//link encoder calibartion data
m_linkEncoderDir :=GVL_CartJointEncoderCaliData.g_asbEncoderDir[i_jntIdx];
m_minLinkEncoder :=GVL_CartJointEncoderCaliData.g_minLinkEncoder[ i_jntIdx] - m_linkEncoderDir*GVL_SetupJointEncoderCaliData.g_linkEncLimitBuffer; // expand limit
m_maxLinkEncoder :=GVL_CartJointEncoderCaliData.g_maxLinkEncoder[ i_jntIdx] + m_linkEncoderDir*GVL_SetupJointEncoderCaliData.g_linkEncLimitBuffer; // expand limit
m_caliLinkEncoder :=GVL_CartJointEncoderCaliData.g_caliLinkEncoder[ i_jntIdx];
m_linkEncCaliJntPos :=GVL_CartJointEncoderCaliData.g_linkEncCaliJntPos[i_jntIdx];
m_linkEncZeroCross :=GVL_CartJointEncoderCaliData.g_linkEncZeroCross[ i_jntIdx];
m_multiCycles :=GVL_CartJointEncoderCaliData.g_multipleCyclesJoint[i_jntIdx];

// convert cali link encoder if joint cross zero
IF 1=m_linkEncZeroCross THEN
	IF 1=m_linkEncoderDir AND m_caliLinkEncoder < m_minLinkEncoder THEN
		m_caliLinkEncoder := GVL_CartJointEncoderCaliData.g_caliLinkEncoder[ i_jntIdx] + m_linkEncoderRes;
	ELSIF -1=m_linkEncoderDir AND m_caliLinkEncoder < m_maxLinkEncoder THEN
		m_caliLinkEncoder := GVL_CartJointEncoderCaliData.g_caliLinkEncoder[ i_jntIdx] + m_linkEncoderRes;
	END_IF
END_IF

// macro data
m_trq2CurrentRatio:=m_motorDir * 1000.0/(m_trqConst*m_motorReduction);
m_current2TrqRatio:=m_motorDir * (m_trqConst*m_motorReduction)/1000.0;
m_linkEnc2PosRatio := 2*PI*m_linkEncoderDir/(m_linkEncoderReduction*m_linkEncoderRes);
m_motorEnc2PosRatio := 2*PI * m_motorDir/(m_motorReduction * m_motorEncoderRes);


// motor data init
m_rawJntVel :=0;
m_curJntVel:=0;
m_curJntTrq :=0;
m_rawCurrent :=0;
m_filtCurrent :=0;
m_cmdJntVel :=0.0;
m_cmdJntTrq :=0.0;
m_cmdCurrent := 0.0;

// filter init
m_jntVelLpf.init(1, GVL_CartControlParameters.g_curJntVelLpfCutoffFreq, g_cartCtrlFreq);
m_cmdTrqLpf.init(1, GVL_CartControlParameters.g_cmdJntTrqLpfCutoffFreq, g_cartCtrlFreq);
m_curTrqLpf.init(1, GVL_CartControlParameters.g_curJntTrqLpfCutoffFreq, g_cartCtrlFreq);

// driver init value
m_motorOutputs.m_controlWord:=DriverCtrlWord_INIT;
m_motorOutputs.m_opMode:=INT_TO_SINT(DriverOPMode_Pos);
m_motorOutputs.m_cmdCurrent:=0;
m_motorOutputs.m_cmdMotorEncoder:=m_motorInputs.m_motorEncoder;
END_METHOD

METHOD PUBLIC updateCmd : BOOL
VAR_INPUT
	i_opMode : E_DriverOPMode;
	i_cmdPos :LREAL;
	i_cmdTrq :LREAL;
	i_cmdVel :LREAL;
END_VAR
VAR
	i:INT;
END_VAR
m_motorOutputs.m_opMode:=INT_TO_SINT( i_opMode);

// pos mode
IF i_opMode = DriverOPMode_Pos OR i_opMode = DriverOPMode_cspMZ  THEN
	m_motorOutputs.m_cmdCurrent:=0;
	m_cmdJntPos :=i_cmdPos;
	m_motorOutputs.m_cmdMotorEncoder :=motorPos2Enc(m_cmdJntPos);
ELSIF i_opMode = DriverOPMode_Vel THEN
	m_cmdJntVel := i_cmdVel;
	m_cartMotorOutput.m_cmdVelMzVelMode := cmd2motorMZ(m_cmdJntVel, g_cartCtrlCycleTime);
ELSIF i_opMode = DriverOPMode_Trq THEN   //Here the torque mode is equal to the contour position mode of the MingZhi driver
	m_cmdJntVel := i_cmdVel;
	m_cmdAcc:=i_cmdVel*2;
	m_cmdJntPos:=i_cmdPos;
	m_cartMotorOutput.m_cmdAccMz :=cmd2motorMZ(m_cmdAcc, g_cartCtrlCycleTime);
	m_cartMotorOutput.m_cmdVelMz := cmd2motorMZ(m_cmdJntVel, g_cartCtrlCycleTime);
	m_motorOutputs.m_cmdMotorEncoder := motorPos2Enc(m_cmdJntVel);
ELSIF i_opMode = DriverOPMode_csvMZ THEN
	m_cmdJntVel := i_cmdVel;
	m_cartMotorOutput.m_cmdVelMzVelMode := cmd2motorMZ(m_cmdJntVel, g_cartCtrlCycleTime);
END_IF
END_METHOD

METHOD PUBLIC updateStatus : BOOL
VAR_INPUT
END_VAR
// compute joint position
m_curLinkPos:= linkEnc2Pos();
m_curMotorPos:=motorEnc2Pos();
m_curLinkSingle := m_curLinkPos - 2*PI* m_linkEncCycles;

// Cart joint1-4 have no link enconder, use motor position
IF m_jntIdx <= 4 THEN
	m_curJntPos := m_curMotorPos;
ELSE
	m_curJntPos := m_curLinkPos;
END_IF

// compute joint velocity
m_curVelCalCycles := m_curVelCalCycles+1;
IF m_curVelCalCycles > m_velCalcCycles THEN
	m_rawJntVel:= (m_curJntPos-m_lastJntPos)/(m_cycleTime*m_velCalcCycles);
	m_curJntVel := m_jntVelLpf.run(m_rawJntVel);
	m_lastJntPos :=m_curJntPos;	
	m_curVelCalCycles:=1;
END_IF


// current and torque
m_rawCurrent := m_motorInputs.m_current;
m_filtCurrent := m_curTrqLpf.run(m_rawCurrent);
m_curJntTrq := m_filtCurrent * m_current2TrqRatio;
END_METHOD

END_FUNCTION_BLOCK

// ---- FBs_Robots/FB_JointBase.TcPOU
FUNCTION_BLOCK FB_JointBase
VAR_INPUT
END_VAR
VAR_OUTPUT
END_VAR
VAR
	// arm and joint index
	m_armIdx :INT;
	m_jntIdx :INT;
	
	// motor IO
	m_motorInputs AT%I*	:ST_MotorInputs;
	m_motorOutputs AT%Q* :ST_MotorOutputs;
	
	// cycle time
	m_cycleTime :LREAL;
	
	// calibrated link encoder data
	m_minLinkEncoder :DINT;
	m_maxLinkEncoder :DINT;
	m_caliLinkEncoder :DINT;
	m_linkEncCaliJntPos :LREAL;
	m_linkEncZeroCross :INT;
	m_initMotorEnc : DINT;
	m_multiCycles :INT;
	
	// joint position from link encoder after power on
	m_initLinkPos :LREAL;
	
	// data for link encoder multiple cycles
	m_lastLinkEncoder :DINT;
	m_linkEncCycles:INT;
	
	// device paramters
	m_motorEncoderRes :DINT;
	m_linkEncoderRes :DINT;
	m_motorReduction :LREAL;
	m_linkEncoderReduction :LREAL;
	m_trqConst :LREAL;
	m_maxCurrent :LREAL;
	m_motorDir :INT;								
	m_linkEncoderDir :INT;
	m_minJntPos: LREAL;
	m_maxJntPos: LREAL;
	
	// macro defined data for quick calculation
	m_trq2CurrentRatio:LREAL;
	m_current2TrqRatio:LREAL;
	m_linkEnc2PosRatio :LREAL;
	m_motorEnc2PosRatio :LREAL;
	
	// joint data
	m_curMotorPos :LREAL;
	m_curLinkPos :LREAL;
	m_curLinkSingle :LREAL;//[0-360]
	m_curJntPos	:LREAL;
	m_curJntVel :LREAL;
	m_rawJntVel :LREAL;
	m_curJntTrq :	LREAL;
	m_rawCurrent : LREAL;
	m_filtCurrent : LREAL;
	m_cmdJntPos :LREAL;
	m_cmdJntVel :LREAL;
	m_cmdJntTrq :LREAL;
	m_cmdCurrent : LREAL;
	m_lastJntPos :LREAL;
	
	// velocity filter
	m_jntVelLpf :FB_LowPassFilter;
	
	// command torque filter
	m_curTrqLpf : FB_LowPassFilter;
	m_cmdTrqLpf :FB_LowPassFilter;
	
	// velocity is calculated every (m_velCalcCycles) control cycles
	// TODO: insturment joint motor can not reach 4k now, so calculate their velocity with 1k frequency, need to remove later
	m_velCalcCycles :INT :=1;
	m_curVelCalCycles :INT :=1;
	
	// SDO writer
	m_opModeSDOWrite:FB_EcCoESdoWrite;
	m_MotorCurrentSDOWrite:FB_EcCoESdoWrite;
	
END_VAR

PROPERTY cmdCurrent : LREAL
GET
cmdCurrent:=m_cmdCurrent;
END_GET
END_PROPERTY

METHOD PUBLIC disable : BOOL
VAR_INPUT
END_VAR
m_motorOutputs.m_controlWord:=DriverCtrlWord_INIT;
disable:=true;
END_METHOD

METHOD PUBLIC enable : BOOL
VAR_INPUT
END_VAR
IF DriverStatusWord_INIT = m_motorInputs.m_statusWord THEN
	m_motorOutputs.m_controlWord:=DriverCtrlWord_PREOP;
	enable := FALSE;
ELSIF DriverStatusWord_PREOP = m_motorInputs.m_statusWord THEN
	m_motorOutputs.m_controlWord:=DriverCtrlWord_OP;
	enable :=  FALSE;
ELSIF DriverStatusWord_OP = m_motorInputs.m_statusWord THEN
	enable :=  TRUE;
//ELSE
//	m_motorOutputs.m_controlWord:=DriverCtrlWord_INIT;
//	enable :=  FALSE;
END_IF
END_METHOD

PROPERTY filtCurrent : LREAL
GET
filtCurrent:=m_filtCurrent;
END_GET
END_PROPERTY

METHOD PUBLIC initJntPos : BOOL
VAR_INPUT
END_VAR
m_lastLinkEncoder :=m_motorInputs.m_linkEncoder;
m_linkEncCycles:=0;
m_curLinkPos :=linkEnc2Pos();
m_initLinkPos:=m_curLinkPos;
m_initMotorEnc :=m_motorInputs.m_motorEncoder;
m_curMotorPos:=motorEnc2Pos();
m_curJntPos := m_curMotorPos;
m_cmdJntPos :=m_curJntPos;	
m_lastJntPos :=m_curJntPos;
END_METHOD

PROPERTY initLinkPos : lreal
GET
initLinkPos:=m_initLinkPos;
END_GET
SET
m_initLinkPos:=initLinkPos;
END_SET
END_PROPERTY

METHOD PUBLIC isEnabled : BOOL
VAR_INPUT
END_VAR
isEnabled :=(DriverStatusWord_OP = m_motorInputs.m_statusWord);
END_METHOD

PROPERTY jntPos : LREAL
GET
jntPos := m_curJntPos;
END_GET
END_PROPERTY

PROPERTY jntTrq : LREAL
GET
jntTrq:=m_curJntTrq;
END_GET
END_PROPERTY

PROPERTY jntVel : LREAL
GET
jntVel := m_curJntVel;
END_GET
END_PROPERTY

METHOD PROTECTED linkEnc2Pos : LREAL
VAR_INPUT
END_VAR
VAR
	incLinkPos :LREAL;
	newLinkEnc :DINT;
END_VAR
// cycle check
IF 1=m_multiCycles THEN
	IF (m_motorInputs.m_linkEncoder - m_lastLinkEncoder)*m_linkEncoderDir < -m_linkEncoderRes/2 THEN
		m_linkEncCycles :=m_linkEncCycles+1;
	ELSIF (m_motorInputs.m_linkEncoder - m_lastLinkEncoder)*m_linkEncoderDir > m_linkEncoderRes/2 THEN
		m_linkEncCycles :=m_linkEncCycles-1;
	END_IF
END_IF
m_lastLinkEncoder:=m_motorInputs.m_linkEncoder;

// convert link encoder if joint cross zero
newLinkEnc := m_motorInputs.m_linkEncoder;
IF 1=m_linkEncZeroCross AND 0 = m_multiCycles THEN
	IF 1=m_linkEncoderDir AND m_motorInputs.m_linkEncoder < m_minLinkEncoder THEN
		newLinkEnc := m_motorInputs.m_linkEncoder + m_linkEncoderRes;
	ELSIF -1=m_linkEncoderDir AND m_motorInputs.m_linkEncoder < m_maxLinkEncoder THEN
		newLinkEnc := m_motorInputs.m_linkEncoder + m_linkEncoderRes;
	END_IF
END_IF

// motion from calibrated points
incLinkPos := (newLinkEnc-m_caliLinkEncoder)*m_linkEnc2PosRatio;

// absolute joint position
linkEnc2Pos := incLinkPos + m_linkEncCaliJntPos + 2*PI* m_linkEncCycles;
END_METHOD

PROPERTY PUBLIC linkPos : LREAL
GET
linkPos:=m_curLinkPos;
END_GET
END_PROPERTY

PROPERTY linkSingle : LREAL
GET
linkSingle :=m_curLinkSingle;
END_GET
END_PROPERTY

METHOD PROTECTED motorEnc2Pos : LREAL
VAR_INPUT
END_VAR
motorEnc2Pos:= (m_motorInputs.m_motorEncoder-m_initMotorEnc)* m_motorEnc2PosRatio +m_initLinkPos;
END_METHOD

PROPERTY PUBLIC motorPos : LREAL
GET
motorPos := m_curMotorPos;
END_GET
END_PROPERTY

METHOD PROTECTED motorPos2Enc : DINT
VAR_INPUT
	i_jntPos :LREAL;
END_VAR

VAR
END_VAR
motorPos2Enc := LREAL_TO_DINT((i_jntPos-m_initLinkPos)/m_motorEnc2PosRatio + m_initMotorEnc);
END_METHOD

PROPERTY rawCurrent : LREAL
GET
rawCurrent := m_rawCurrent;
END_GET
END_PROPERTY

METHOD PROTECTED singleCyclePos : LREal
VAR_INPUT
END_VAR
VAR
	cycles :lreal;
END_VAR
cycles := ABS(FLOOR( m_curJntPos/g_2pi));
IF m_curJntPos<0 THEN
	singleCyclePos := m_curJntPos+cycles*g_2pi;
ELSE
	singleCyclePos := m_curJntPos-cycles*g_2pi;
END_IF
END_METHOD

METHOD PUBLIC updateCmds : BOOL
VAR_INPUT
	i_opMode : E_DriverOPMode;
	i_cmdPos :LREAL;
	i_cmdTrq :LREAL;
END_VAR
VAR
	filtCmdTrq :LREAL;
END_VAR
m_motorOutputs.m_opMode:=INT_TO_SINT( i_opMode);
// pos mode
IF i_opMode = DriverOPMode_Pos THEN
	m_motorOutputs.m_cmdCurrent:=0;
	m_cmdTrqLpf.reset();	
//	i_cmdPos:=LIMIT(m_minJntPos, i_cmdPos, m_maxJntPos); // May cause position jump, Do this in safety check. 
	m_cmdJntPos :=i_cmdPos;
	m_motorOutputs.m_cmdMotorEncoder :=motorPos2Enc(m_cmdJntPos);
ELSIF i_opMode = DriverOPMode_Trq THEN
	filtCmdTrq:=m_cmdTrqLpf.run(i_cmdTrq);
	m_motorOutputs.m_cmdCurrent:=LREAL_TO_DINT(LIMIT(-m_maxCurrent, filtCmdTrq*m_trq2CurrentRatio,m_maxCurrent));
	m_motorOutputs.m_cmdMotorEncoder :=m_motorInputs.m_motorEncoder; 
END_IF
m_cmdCurrent:=m_motorOutputs.m_cmdCurrent;
END_METHOD

METHOD PUBLIC updateStatus : BOOL
VAR_INPUT
END_VAR
// compute joint position
m_curLinkPos:= linkEnc2Pos();
m_curMotorPos:=motorEnc2Pos();
m_curJntPos := m_curMotorPos;
m_curLinkSingle := singleCyclePos();

// compute joint velocity
m_curVelCalCycles := m_curVelCalCycles+1;
IF m_curVelCalCycles > m_velCalcCycles THEN
	m_rawJntVel:= (m_curJntPos-m_lastJntPos)/(m_cycleTime*m_velCalcCycles);
	m_curJntVel := m_jntVelLpf.run(m_rawJntVel);
	m_lastJntPos :=m_curJntPos;	
	m_curVelCalCycles:=1;
END_IF


// current and torque
m_rawCurrent := m_motorInputs.m_current;
m_filtCurrent := m_curTrqLpf.run(m_rawCurrent);
m_curJntTrq := m_filtCurrent * m_current2TrqRatio;
END_METHOD

END_FUNCTION_BLOCK

// ---- FBs_CartControlles/FB_CartCtrlMotionCar.TcPOU
FUNCTION_BLOCK FB_CartCtrlMotionCar EXTENDS FB_CartCtrlBase
VAR_INPUT
END_VAR
VAR_OUTPUT
END_VAR
VAR
	m_driveForce: ARRAY [1..2] OF LREAL;
	
	// input drive force filter
	m_driveVelLpf : ARRAY [1..2] OF FB_LowPassFilter;
	m_driveForceFilter: Vec2i;
	
	//cart motion trajectory velocity
	m_trajVel : ARRAY [1..2] OF LREAL;
	m_motorDir :ARRAY [1..2] OF INT := [1,-1];
	
	m_tarJntPos : ARRAY [1..2] OF LREAL;
	m_incJntPos : ARRAY [1..2] OF LREAL;
	m_initJntPos : ARRAY [1..2] OF LREAL;
	// time threshold to drive wheel after it's enabled
	m_cartWheelDriveWaitTime :LREAL := 0.2;
	
	//wheel motion  time 
	m_wheelMotionTime:ARRAY [1..2] OF LREAL;
	
	// filter cut-off frequency for cart drive force 
	m_cmdJntVelLpfCutoffFreq : LREAL :=5;
END_VAR

VAR CONSTANT
	//Proportionality constant of force sensor
	m_driveForceProConstant : LREAL := 5/15000;
END_VAR

// override this function in each exact controller
METHOD PROTECTED calcCmdJntPos : BOOL
VAR_IN_OUT CONSTANT
	// slave cart joint data
	i_slaveCart :FB_SlaveCart;
END_VAR

VAR
	i:INT;
END_VAR

FOR i := 1 TO 2 BY 1 DO
	m_driveForce[i] :=LIMIT(-5, i_slaveCart.m_driveForce[i]/3000, 5);
	m_wheelMotionTime[i] := LIMIT(0, m_wheelMotionTime[i] + g_cartCtrlCycleTime, 1);
	
	IF m_wheelMotionTime[i] > m_cartWheelDriveWaitTime THEN
		m_trajVel[i] := m_driveVelLpf[i].run(i_rawData:=m_motorDir[i] * m_driveForce[i]/2);
		m_incJntPos[i] := m_incJntPos[i] + m_trajVel[i] * g_cartCtrlCycleTime;
		
		m_cmdJntPos[i+2] := m_initJntPos[i] + m_incJntPos[i];
	END_IF
END_FOR
END_METHOD

// override this function in each exact controller
// NOTICE: set joint control mode here, and do some initialization if needed
METHOD PUBLIC init : BOOL
VAR_IN_OUT CONSTANT
	i_slaveCart	:FB_SlaveCart;
END_VAR
VAR_IN_OUT 
	r_cartCtrlCmd :ST_SlaveArmCtrlCmds;
END_VAR
SUPER^.init(i_slaveCart,r_cartCtrlCmd);

m_jntEnableFlag[3] :=1;
m_jntEnableFlag[4] :=1;

m_jntOPMode[3]:= DriverOPMode_cspMZ;
m_jntOPMode[4]:= DriverOPMode_cspMZ;

m_tarJntPos[1] := 0;
m_tarJntPos[2] := 0;

m_incJntPos[1] := 0;
m_incJntPos[2] := 0;

m_initJntPos[1] := i_slaveCart.curJntPos[3];
m_initJntPos[2] := i_slaveCart.curJntPos[4];

m_driveVelLpf[1].init(i_filterOrd:= 1, i_cutoffFreq:= m_cmdJntVelLpfCutoffFreq, i_sampleFreq:= 8000);
m_driveVelLpf[2].init(i_filterOrd:= 1, i_cutoffFreq:= m_cmdJntVelLpfCutoffFreq, i_sampleFreq:= 8000);

m_driveVelLpf[1].run(i_rawData:=0);
m_driveVelLpf[2].run(i_rawData:=0);


m_wheelMotionTime[1]:=0;
m_wheelMotionTime[2]:=0;

// update commands to arm
copyCmds(r_cartCtrlCmd);
END_METHOD

END_FUNCTION_BLOCK

// ---- FBs_CartControlles/FB_CartCtrlAdjust.TcPOU
FUNCTION_BLOCK FB_CartCtrlAdjust EXTENDS FB_CartCtrlBase
VAR_INPUT
END_VAR
VAR_OUTPUT
END_VAR
VAR

	m_joystickSignal: Vec8d;	
	m_fiducialValue:INT:= 512;
	m_joystickRange:INT:=430;
	m_joystickDir: Vec8i:=[1,1,1,1,-1,-1,1,-1];
	m_joystickVelInc: Vec8d;
	m_actJntPos: Vec8d;
	m_tarPosInc: Vec8d;
	m_tarCartPos: Vec8d;
	m_trajJntPos : Vec8d;
	m_tarJntPos : Vec8d;
	m_initActJntPos: Vec8d;
	m_initActCartPos: Vec8d;
	m_veiwAngle : LREAL;

	m_carJntSoftwareLimit :ARRAY [5..8] OF LREAL := [0.005, 2*g_deg2Rad, 0.005, 2*g_deg2Rad];
	// input joystick signal filter
	m_joystickSignalLpf : ARRAY [1..4] OF FB_LowPassFilter;
	m_joystickSignalFilter: Vec8d;
	
	// time threshold to 5-8joint after it's enabled
	m_cartAdjustStartWaitTime :LREAL := 0.2;
	
	//adjust start  time 
	m_adjustStartTime :LREAL;
	
	// filter cut-off frequency for cart drive force 
	m_cmdJoystickLpfCutoffFreq : LREAL :=8;
	m_cartCtrlFreq :LREAL:=8000;
	
	m_jntOTG :ARRAY[1..8] OF FB_secOrdTrajFilter;
END_VAR

// override this function in each exact controller
METHOD PROTECTED calcCmdJntPos : BOOL
VAR_IN_OUT CONSTANT
	// slave cart joint data
	i_slaveCart :FB_SlaveCart;
END_VAR

VAR
	i:INT;
END_VAR
//In this method, 5 represents the pillar postion , 6 represents the beam rotation angle ,7 represents the beam stretch position ,8 represents the overhang angle
m_adjustStartTime :=LIMIT(0, m_adjustStartTime + g_cartCtrlCycleTime, 1);
m_actJntPos := i_slaveCart.curJntPos;
m_actJntPos[7] := i_slaveCart.curJntPos[7] + GVL_CartControlParameters.g_curBeamStretchJntInitPos;
m_veiwAngle := m_actJntPos[6] + m_actJntPos[8];

IF m_adjustStartTime > m_cartAdjustStartWaitTime THEN
	FOR i:= 1 TO 4 BY 1 DO
		m_joystickSignalFilter[i] := m_joystickSignalLpf[i].run(i_rawData:= m_joystickSignal[i]);
		m_joystickSignal[i] := i_slaveCart.m_joystickSignal[i] - m_fiducialValue;
		m_joystickVelInc[i+4] := m_joystickSignalFilter[i]/m_joystickRange*m_joystickDir[i+4]*GVL_CartControlParameters.g_maxCartVel[i];
		m_tarPosInc[i+4] := m_tarPosInc[i+4] + m_joystickVelInc[i+4] * g_cartCtrlCycleTime;
	END_FOR
	
	
	m_tarCartPos[5] := m_initActJntPos[5] + m_tarPosInc[5];
	IF i_slaveCart.m_ctrlEnable.camera_joysticks_enable THEN
		m_tarCartPos[6] := m_initActCartPos[6] + m_tarPosInc[6]*COS(m_veiwAngle)+m_tarPosInc[7]*SIN(m_veiwAngle);
		m_tarCartPos[7] := m_initActCartPos[7] - m_tarPosInc[6]*SIN(m_veiwAngle)+m_tarPosInc[7]*COS(m_veiwAngle);
	ELSE
		m_tarCartPos[6] := m_initActCartPos[6] + m_tarPosInc[6];
		m_tarCartPos[7] := m_initActCartPos[7] + m_tarPosInc[7];
	END_IF
	m_tarCartPos[8] := m_initActJntPos[8] + m_tarPosInc[8];
	
	IF i_slaveCart.m_ctrlEnable.limit_height_adjusting THEN
		m_trajJntPos[5] := m_tarCartPos[5];
	ELSE
		m_trajJntPos[5] := LIMIT(GVL_CartMotorParameters.g_minJntPos[5], m_tarCartPos[5], MAX(m_actJntPos[5],i_slaveCart.m_cartDataFromUI.m_standColumnHightLimit));
	END_IF
	m_trajJntPos[6] := atan2( m_tarCartPos[6], m_tarCartPos[7]);
	m_trajJntPos[7] := m_tarCartPos[7]/COS(m_trajJntPos[6]) - GVL_CartControlParameters.g_curBeamStretchJntInitPos;
	m_trajJntPos[8] := m_tarCartPos[8] -  (m_trajJntPos[6] - m_initActJntPos[6]);
	
	
	
	m_tarJntPos[5] := LIMIT(GVL_CartMotorParameters.g_minJntPos[5] + m_carJntSoftwareLimit[5], m_trajJntPos[5], GVL_CartMotorParameters.g_maxJntPos[5] - m_carJntSoftwareLimit[5]) ;
	m_tarJntPos[6] := LIMIT(GVL_CartMotorParameters.g_minJntPos[6] + m_carJntSoftwareLimit[6], m_trajJntPos[6], GVL_CartMotorParameters.g_maxJntPos[6] - m_carJntSoftwareLimit[6]);
	m_tarJntPos[7] := LIMIT(GVL_CartMotorParameters.g_minJntPos[7] + m_carJntSoftwareLimit[7], m_trajJntPos[7], GVL_CartMotorParameters.g_maxJntPos[7] - m_carJntSoftwareLimit[7]);
	m_tarJntPos[8] := LIMIT(GVL_CartMotorParameters.g_minJntPos[8] + m_carJntSoftwareLimit[8], m_trajJntPos[8], GVL_CartMotorParameters.g_maxJntPos[8] - m_carJntSoftwareLimit[8]);
	
	FOR i := 5 TO 8 BY 1 DO
		m_jntOTG[i].run(i_targetPos:= m_tarJntPos[i], i_targetVel:= 0.0, o_cmdAcc=> , o_cmdVel=> , o_cmdPos=>m_cmdJntPos[i] );
	END_FOR
END_IF
END_METHOD

// override this function in each exact controller
// NOTICE: set joint control mode here, and do some initialization if needed
METHOD PUBLIC init : BOOL
VAR_IN_OUT CONSTANT
	i_slaveCart	:FB_SlaveCart;
END_VAR
VAR_IN_OUT 
	r_cartCtrlCmd :ST_SlaveArmCtrlCmds;
END_VAR
VAR
	i:INT;
END_VAR
// check if to hold the command joint position unchanged
//m_holdLastCmds := checkToHoldLastCmds(i_slaveCart);

SUPER^.init(i_slaveCart,r_cartCtrlCmd);

m_jntEnableFlag[5] :=1;
m_jntEnableFlag[6] :=1;
m_jntEnableFlag[7] :=1;
m_jntEnableFlag[8] :=1;

m_jntOPMode[5]:= DriverOPMode_cspMZ;
m_jntOPMode[6]:= DriverOPMode_Pos;
m_jntOPMode[7]:= DriverOPMode_Pos;
m_jntOPMode[8]:= DriverOPMode_Pos;

m_joystickSignalFilter := g_zeroVec8d;
m_joystickSignal := g_zeroVec8d;
m_tarPosInc := g_zeroVec8d;
m_trajJntPos := g_zeroVec8d;

m_initActJntPos:=i_slaveCart.curJntPos;
m_initActCartPos[6] := (m_initActJntPos[7] + GVL_CartControlParameters.g_curBeamStretchJntInitPos) * SIN(m_initActJntPos[6]);
m_initActCartPos[7] := (m_initActJntPos[7] + GVL_CartControlParameters.g_curBeamStretchJntInitPos) * COS(m_initActJntPos[6]);

FOR i := 1 TO 4 BY 1 DO
	m_jntOTG[i+4].init(i_curCmdPos:= m_cmdJntPos[i+4], i_curCmdVel:= 0, i_maxV:=GVL_CartControlParameters.g_maxJntVel[i+4] , i_maxA:=GVL_CartControlParameters.g_maxJntAcc[i+4] , i_Ts:=g_cartCtrlCycleTime );
	m_joystickSignalLpf[i].init(i_filterOrd:= 1, i_cutoffFreq:= m_cmdJoystickLpfCutoffFreq, i_sampleFreq:= m_cartCtrlFreq);
END_FOR

m_adjustStartTime := 0;
// update commands to arm
copyCmds(r_cartCtrlCmd);
END_METHOD

END_FUNCTION_BLOCK

// ---- FBs_CartControlles/FB_CartCtrlInSurgery.TcPOU
FUNCTION_BLOCK FB_CartCtrlInSurgery EXTENDS FB_CartCtrlBase
VAR_INPUT
END_VAR
VAR_OUTPUT
END_VAR
VAR
END_VAR

// override this function in each exact controller
METHOD PROTECTED calcCmdJntPos : BOOL
VAR_IN_OUT CONSTANT
	// slave cart joint data
	i_slaveCart :FB_SlaveCart;
END_VAR
m_cmdJntPos := i_slaveCart.curJntPos;
END_METHOD

// override this function in each exact controller
// NOTICE: set joint control mode here, and do some initialization if needed
METHOD PUBLIC init : BOOL
VAR_IN_OUT CONSTANT
	i_slaveCart	:FB_SlaveCart;
END_VAR
VAR_IN_OUT 
	r_cartCtrlCmd :ST_SlaveArmCtrlCmds;
END_VAR
SUPER^.init(i_slaveCart,r_cartCtrlCmd);

// update commands to arm
copyCmds(r_cartCtrlCmd);
END_METHOD

END_FUNCTION_BLOCK

// ---- FBs_RobotDynamics/FB_SetupGravity.TcPOU
FUNCTION_BLOCK FB_SetupGravity
VAR_INPUT
END_VAR
VAR
	m_armIdx :INT ;

	// current arm parameters
	m_armParams :ARRAY[1..7] OF LREAL;

	// gravity regression matrix
	regMat:ARRAY[1..7] OF LREAL;
	
	m_graivty :LREAL;
END_VAR

METHOD getRegMat : BOOL
VAR_INPUT
	// joint position of setup joint, joint6-8
	setupAng :LREAL;
	q1: LREAL;
	q2: LREAL;
	q3: LREAL;
END_VAR

VAR
	s0,c0,s1,c1,s2, c2,d3 :LREAL;
END_VAR

VAR_OUTPUT
	o_regMat:ARRAY[1..7] OF LREAL;
END_VAR
s0:= SIN(setUpAng);
c0:= COS(setUpAng);
s1:=SIN(q1);
c1:=COS(q1);
s2:=SIN(q2);
c2:=COS(q2);
d3:=q3;

// setup joint
o_regMat[1] :=c0;
o_regMat[2] := s0;
o_regMat[3] :=-(c2*s0*d3+c0*c1*s2*d3);
o_regMat[4] :=  -c0*c1;
o_regMat[5] :=  -c0*s1;
o_regMat[6] := - (c0*c1*s2+c2*s0);
o_regMat[7] :=  s0*s2- c0*c1*c2  ;
END_METHOD

METHOD init : BOOL
VAR_INPUT
	i_armIdx :INT;
END_VAR
m_armIdx :=i_armIdx;
END_METHOD

METHOD run : BOOL
VAR_IN_OUT CONSTANT
	// setup joint angle
	i_setupJntPos :Vec5d;
	
	// slave joint angle
	i_slaveJntPos :Vec8d;
	
	// instrument
	i_instruStatus :ST_InstruStatus;
END_VAR
VAR_OUTPUT
	// setup joint3 gravity
	o_jnt3Gravity :LREAL;
	
	// setup joint5 gravity
	o_jnt5Gravity :LREAL;
END_VAR
VAR
	setupPos, q1, q2, q3 :LREAL;
	i,j:INT;
	
	gravityTrq :Vec4d;

END_VAR
setupPos:=i_setupJntPos[5];
q1 := i_slaveJntPos[1];
q2 := i_slaveJntPos[2];
q3 := i_slaveJntPos[3];

// get regression matrx
getRegMat(setupPos, q1, q2, q3, o_regMat=>regMat);

// determine current arm parameters
m_armParams[1] := GVLs_SetupArmDynamics.g_setupJnt5GravityParam[m_armIdx,1];
m_armParams[2] := GVLs_SetupArmDynamics.g_setupJnt5GravityParam[m_armIdx,2];
IF FALSE = i_instruStatus.m_ready THEN
	// arm only
	FOR i:=1 TO 5 DO
		m_armParams[i+2]:=g_gravityParam[m_armIdx,i];
	END_FOR

// endoscope
ELSIF InstruType_endoscope = i_instruStatus.m_type THEN 
	FOR i:=1 TO 5 DO
		m_armParams[i+2]:=g_gravityParam[m_armIdx,i]+g_gravityEndoscope[i];
	END_FOR

// instrument
ELSE
	FOR i:=1 TO 5 DO
		m_armParams[i+2]:=g_gravityParam[m_armIdx,i]+g_gravityInstrument[i];
	END_FOR
// TODO:Trocar
END_IF

// calculate gravity torque
o_jnt5Gravity:=0;
FOR j:=1 TO 7 DO
	o_jnt5Gravity:=o_jnt5Gravity+regMat[j]*m_armParams[j];
END_FOR
m_graivty := o_jnt5Gravity;

o_jnt3Gravity:= setupJnt3Gravity(i_setupJntPos[3]);
END_METHOD

METHOD setupJnt3Gravity : LREAL
VAR_INPUT
	i_jnt3Pos :LREAL;
END_VAR
VAR
	q:LREAL;
END_VAR
q := LIMIT(g_setupJnt3GravityPosRange[m_armIdx,1], i_jnt3Pos, g_setupJnt3GravityPosRange[m_armIdx,2]);
setupJnt3Gravity:=g_setupJnt3GravityParams[m_armIdx,1]*EXPT(q,3)+g_setupJnt3GravityParams[m_armIdx,2]*EXPT(q,2)+
				g_setupJnt3GravityParams[m_armIdx,3]*q+g_setupJnt3GravityParams[m_armIdx,4];
END_METHOD

END_FUNCTION_BLOCK

// ---- FBs_Robots/FB_SetupArm.TcPOU
FUNCTION_BLOCK FB_SetupArm
VAR_INPUT
END_VAR
VAR_OUTPUT
END_VAR
VAR
	// arm index, from 1 to 4
	m_armIdx: INT;
	
	// joints
	m_joints :ARRAY[1..g_setupJntNum] OF FB_SetupJoint;
	
	// adjust detect
	m_adjustIO AT%I* :UDINT;
	m_manualAdjustOnFlag :BOOL;
	m_jnt5AdjustDir :INT; // -1, 0, 1;
	m_manualAdjustDetect : FB_setupAdjustDetect;
	m_jnt5AdjustDetect : FB_setupJnt5AdjustDetect;
	
	// arm cartesian data, defined in cart origin
	m_curCartPose	:ST_Frame;
	
	// cartesion position of remote center
	m_rcPos :Vec3d;	
	
	// arm joint data
	m_curMotorPos :Vec5d;
	m_curLinkPos :Vec5d;
	m_curJntPos :Vec5d;
	m_curJntVel :Vec5d;
	m_curJntTrq :Vec5d;
	m_rawJntCurrent :Vec5d;
	m_filtJntCurrent :Vec5d;
	m_cmdJntCurrent : Vec5d;
	m_cmdJntPos :Vec5d;
	m_cmdJntVel :Vec5d;
	m_cmdJntTrq :Vec5d;
		
	// arm gravity
	m_jntGravity : Vec5d:=g_zeroVec5d;
	
	// joint position controller
	m_jntPIDCtrl :ARRAY[1..g_setupJntNum] OF FB_PID;
	
END_VAR

PROPERTY armIdx : int
GET
armIdx:=m_armIdx;
END_GET
END_PROPERTY

METHOD PROTECTED checkIO : BOOL
VAR_INPUT
END_VAR
// check manual and auto adjust button
m_manualAdjustOnFlag := m_manualAdjustDetect.run(m_adjustIO);
m_jnt5AdjustDir := m_jnt5AdjustDetect.run(m_adjustIO);
END_METHOD

PROPERTY cmdJntCurrent : REFERENCE TO  Vec5d
GET
cmdJntCurrent ref= m_cmdJntCurrent;
END_GET
END_PROPERTY

PROPERTY curCartPose : REFERENCE TO ST_Frame
GET
curCartPose ref=m_curCartPose;
END_GET
END_PROPERTY

PROPERTY curJntPos : REFERENCE TO Vec5d
GET
curJntPos ref=m_curJntPos;
END_GET
END_PROPERTY

PROPERTY curJntTrq : REFERENCE TO Vec5d
GET
curJntTrq ref=m_curJntTrq;
END_GET
END_PROPERTY

PROPERTY curJntVel :REFERENCE TO Vec5d
GET
curJntVel ref=m_curJntVel;
END_GET
END_PROPERTY

PROPERTY curLinkPos :REFERENCE TO Vec5d
GET
curLinkPos ref=m_curLinkPos;
END_GET
END_PROPERTY

PROPERTY curMotorPos : REFERENCE TO  Vec5d
GET
curMotorPos ref=m_curMotorPos;
END_GET
END_PROPERTY

METHOD PUBLIC enable : BOOL
VAR_IN_OUT CONSTANT
	i_jntIdx :Vec5i;
END_VAR
VAR
	i :INT ;
END_VAR
FOR i:=1 TO g_setupJntNum DO
	IF 1= i_jntIdx[i] THEN
		m_joints[i].enable();
	ELSE
		m_joints[i].disable();
	END_IF
END_FOR
END_METHOD

PROPERTY filtJntCurrent :REFERENCE TO Vec5d
GET
filtJntCurrent ref= m_filtJntCurrent;
END_GET
END_PROPERTY

// compute cartesion pose in cart origin
METHOD PROTECTED forwardKinematic : BOOL
VAR_IN_OUT CONSTANT
	i_jntPos :Vec5d;
END_VAR
VAR_IN_OUT
	r_cartPose :ST_Frame;
	
	// position of remote center
	r_rcPos :Vec3d;
END_VAR
VAR
	a2,d4,d6:LREAL; //DH parameters
	
	Radius,Angle,R1,q:LREAL; //Disk structure parameters
	x,y,z:LREAL;
	basePosMatrix:ARRAY[1..4,1..4] OF LREAL;//transform from origin to C0
	
	T_50:ARRAY[1..4,1..4] OF LREAL; //transform from C0 to C5
	F5:ARRAY[1..4,1..4] OF LREAL; //transform from origin to C5
	q1,q2,q3,q4,q5:LREAL;	
	c14,s14,c5,s5,s1,c1:LREAL;
	
	fixPointTransform:ARRAY[1..4,1..4] OF LREAL; //transform from C5 to fixed point
	fixPointMatrix:ARRAY[1..4,1..4] OF LREAL;
END_VAR
//TODO: move DH parameter to GVL 


//****************input:five joint position of SetupArm********************//
q1:=i_jntPos[1]; q2:=i_jntPos[2]; q3:=i_jntPos[3]; q4:=i_jntPos[4]; q5:=i_jntPos[5];

//**********************DH parameters*************************//
IF (m_armIdx=1) THEN
	a2:=0.019; d4:=0.3545;
	
ELSIF (m_armIdx=2) THEN
	a2:=0.136; d4:=0.3545;
	
ELSIF (m_armIdx=3) THEN	
	a2:=0.136; d4:=0.5205;
	
ELSIF (m_armIdx=4) THEN	
	a2:=0.1825; d4:=0.5205;
END_IF
d6:=0.6387229+0.1659;

//********************transform form origin to C0***********************//
Radius:=0.170; Angle:=60.0*g_deg2Rad;
R1:=Radius;  q:=Angle;
IF (m_armIdx=1) THEN
	x:=-R1; y:=0; z:=0;
	
ELSIF (m_armIdx=2) THEN
	x:=-R1*COS(q); y:=-R1*SIN(q); z:=0;
	
ELSIF (m_armIdx=3) THEN	
	x:=R1*COS(q); y:=-R1*SIN(q); z:=0;
	
ELSIF (m_armIdx=4) THEN	
	x:=R1; y:=0; z:=0;
END_IF

basePosMatrix[1,1]:=0;
basePosMatrix[2,1]:=1;
basePosMatrix[3,1]:=0;
basePosMatrix[4,1]:=0;

basePosMatrix[1,2]:=-1;
basePosMatrix[2,2]:=0;
basePosMatrix[3,2]:=0;
basePosMatrix[4,2]:=0;

basePosMatrix[1,3]:=0;
basePosMatrix[2,3]:=0;
basePosMatrix[3,3]:=1;
basePosMatrix[4,3]:=0;

basePosMatrix[1,4]:=x;
basePosMatrix[2,4]:=y;
basePosMatrix[3,4]:=z;
basePosMatrix[4,4]:=1;

//***************output1:C5 posture relative to origin(other than C0)*************//
c14:=COS(q1+q4); s14:=SIN(q1+q4); 
c5:=COS(q5); s5:=SIN(q5);
c1:=COS(q1); s1:=SIN(q1);

T_50[1,1]:=c14*c5; 
T_50[2,1]:=s14*c5; 
T_50[3,1]:=-s5; 
T_50[4,1]:=0;

T_50[1,2]:=-c14*s5;
T_50[2,2]:=-s14*s5; 
T_50[3,2]:=-c5; 
T_50[4,2]:=0;

T_50[1,3]:=-s14;
T_50[2,3]:=c14;
T_50[3,3]:=0;
T_50[4,3]:=0;

T_50[1,4]:=a2*c1 + q2*s1;
T_50[2,4]:=a2*s1 - q2*c1;
T_50[3,4]:=d4 + q3;
T_50[4,4]:=1;

matMultiply(basePosMatrix,T_50,F5);
r_cartPose.m_pos[1]:=F5[1,4]; r_cartPose.m_pos[2]:=F5[2,4]; r_cartPose.m_pos[3]:=F5[3,4];

r_cartPose.m_rot[1,1]:=F5[1,1];  r_cartPose.m_rot[1,2]:=F5[1,2];  r_cartPose.m_rot[1,3]:=F5[1,3];
r_cartPose.m_rot[2,1]:=F5[2,1];  r_cartPose.m_rot[2,2]:=F5[2,2];  r_cartPose.m_rot[2,3]:=F5[2,3];
r_cartPose.m_rot[3,1]:=F5[3,1];  r_cartPose.m_rot[3,2]:=F5[3,2];  r_cartPose.m_rot[3,3]:=F5[3,3];

//********************output2:remote center position************************//
fixPointTransform[1,1]:=1;  fixPointTransform[2,2]:=1;  fixPointTransform[3,3]:=1;  fixPointTransform[4,4]:=1;  
fixPointTransform[2,4]:=-d6;  
matMultiply(F5,fixPointTransform,fixPointMatrix);
r_rcPos[1]:=fixPointMatrix[1,4];  r_rcPos[2]:=fixPointMatrix[2,4];  r_rcPos[3]:=fixPointMatrix[3,4];
END_METHOD

METHOD PUBLIC init : BOOL
VAR_INPUT
	i_armIdx:INT;
END_VAR
VAR 
	i :INT ;
	currentRatioMotor2Jnt:LREAL;
END_VAR
// arm statues init
m_armIdx:=i_armIdx;

// joint init
FOR i:=1 TO g_setupJntNum DO
	m_joints[i].init(m_armIdx, i,g_setupArmCtrlCycleTime);
END_FOR

// joint init
FOR i:=1 TO g_setupJntNum DO
	m_joints[i].initJntPos();
END_FOR

// update arm status if joint position is re-init
updateStatus();

// joint controller init
FOR i:=1 TO g_setupJntNum DO 
	currentRatioMotor2Jnt:=GVL_SetupMotorParameters.g_motorTrqConst[i]*GVL_SetupMotorParameters.g_motorReduction[i]/1000;
	m_jntPIDCtrl[i].init(g_setupArmCtrlCycleTime,GVL_SetupControlParameters.g_posKp[i],GVL_SetupControlParameters.g_posKd[i],
		GVL_SetupControlParameters.g_posKi[i], GVL_SetupControlParameters.g_posKiLimit[i]* currentRatioMotor2Jnt,
		GVL_SetupControlParameters.g_posCtrlLimit[i]*currentRatioMotor2Jnt);
END_FOR
END_METHOD

METHOD PUBLIC isEnabled : BOOL
VAR_IN_OUT CONSTANT
	i_jntIdx :Vec5i;
END_VAR
VAR
	i :INT ;
END_VAR
isEnabled := TRUE;
FOR i:=1 TO g_setupJntNum DO
	IF 1= i_jntIdx[i] THEN
		isEnabled :=  (m_joints[i].isEnabled() AND isEnabled);
	END_IF
END_FOR
END_METHOD

PROPERTY jnt5AdjustDir : int
GET
jnt5AdjustDir := m_jnt5AdjustDir;
END_GET
END_PROPERTY

PROPERTY jntGravity :REFERENCE TO Vec5d
GET
jntGravity ref=m_jntGravity;
END_GET
END_PROPERTY

PROPERTY manualAdjustOn : bool
GET
manualAdjustOn := m_manualAdjustOnFlag;
END_GET
END_PROPERTY

PROPERTY rawJntCurrent :REFERENCE TO Vec5d
GET
rawJntCurrent ref=m_rawJntCurrent;
END_GET
END_PROPERTY

PROPERTY rcPos :REFERENCE to Vec3d
GET
rcPos REF= m_rcPos;
END_GET
END_PROPERTY

// update joints control command
METHOD PUBLIC updateCmds : BOOL
VAR_IN_OUT CONSTANT
	i_armCtrlCmd : ST_SetupArmCtrlCmds;
END_VAR
VAR
	i:INT;
END_VAR
m_cmdJntTrq:=i_armCtrlCmd.m_cmdJntTrq;
m_cmdJntPos :=i_armCtrlCmd.m_cmdJntPos;
m_cmdJntVel :=i_armCtrlCmd.m_cmdJntVel;

// enable/disable joints
enable(i_armCtrlCmd.m_jntEnableFlag);

// position/torque control
FOR i:=1 TO g_setupJntNum DO 
	IF i_armCtrlCmd.m_jntOPMode[i]=DriverOPMode_PosTrq THEN
		// position controller and gravity feedforward
		m_cmdJntTrq[i]:=m_jntPIDCtrl[i].run(m_cmdJntPos[i],m_curJntPos[i],0,m_curJntVel[i]);
		m_cmdJntTrq[i]:=m_cmdJntTrq[i]+m_jntGravity[i];
		m_joints[i].updateCmds(DriverOPMode_Trq,m_cmdJntPos[i],m_cmdJntTrq[i]);
	ELSIF i_armCtrlCmd.m_jntOPMode[i]=DriverOPMode_Trq THEN
		// gravity feedforward
		m_jntPIDCtrl[i].reset();
		m_cmdJntTrq[i]:=m_cmdJntTrq[i]+m_jntGravity[i]+GVLs_SetupArmDynamics.g_setupJntGravityOffset[m_armIdx, i];
		m_joints[i].updateCmds(DriverOPMode_Trq,i_armCtrlCmd.m_cmdJntPos[i],m_cmdJntTrq[i]);
	ELSE
		m_jntPIDCtrl[i].reset();
		m_cmdJntTrq[i]:=0;
		m_joints[i].updateCmds(DriverOPMode_Pos,i_armCtrlCmd.m_cmdJntPos[i],m_cmdJntTrq[i]);
	END_IF
	
END_FOR
END_METHOD

METHOD PUBLIC updateDyna : BOOL
VAR_IN_out constant
	i_jnt3Gravity :LREAL;
	i_jnt5Gravity :LREAL;
END_VAR
m_jntGravity[3]:=i_jnt3Gravity;
m_jntGravity[5]:=i_jnt5Gravity;
END_METHOD

// update arm status, including kinematic and dynamic
METHOD PUBLIC updateStatus : BOOL
VAR_INPUT
END_VAR
VAR 
	i,j:INT;
END_VAR
// update joint data
FOR i:=1 TO g_setupJntNum DO
	m_joints[i].updateStatus();
END_FOR

// check adjust button
checkIO();

// get joint data
FOR i:=1 TO g_setupJntNum DO
	m_curMotorPos[i]:=m_joints[i].motorPos;
	m_curLinkPos[i]:=m_joints[i].linkPos;
	m_curJntPos[i]:=m_joints[i].jntPos;
	m_curJntVel[i]:=m_joints[i].jntVel;
	m_curJntTrq[i]:=m_joints[i].jntTrq;
	m_rawJntCurrent[i]:=m_joints[i].rawCurrent;
	m_filtJntCurrent[i]:=m_joints[i].filtCurrent;
	m_cmdJntCurrent[i]:=m_joints[i].cmdCurrent;
END_FOR 

// cartesion pose
forwardKinematic(m_curJntPos,m_curCartPose,m_rcPos);
END_METHOD

END_FUNCTION_BLOCK

// ---- FBs_Robots/FB_SetupRobot.TcPOU
FUNCTION_BLOCK FB_SetupRobot
VAR_INPUT
END_VAR
VAR_OUTPUT
END_VAR
VAR
	// setup arms, responsible for arm kinematic and control
	m_setupArms :ARRAY[1..g_sArmNum] OF FB_SetupArm;
	
	// arm state
	m_setupArmState:ARRAY[1..g_sArmNum] OF E_setupArmState:=[4(E_setupArmState.SetupArmState_Error)];
	m_lastSetupArmState:ARRAY[1..g_sArmNum] OF E_setupArmState:=[4(E_setupArmState.SetupArmState_Error)];
	m_nextSetupArmState:ARRAY[1..g_sArmNum] OF E_setupArmState:=[4(E_setupArmState.SetupArmState_Error)];
	
	// all arm controller instance 
	m_armCtrlFactory :ARRAY[1..g_sArmNum,1..SetupArmState_totalNum] OF I_SetupArmCtrl;
	m_armInit :ARRAY[1..g_sArmNum] OF FB_SetupCtrlInit;
	m_armError :ARRAY[1..g_sArmNum] OF FB_SetupCtrlError;
	m_armSelfCheck :ARRAY[1..g_sArmNum] OF FB_SetupCtrlSelfCheck;
	m_armHold :ARRAY[1..g_sArmNum] OF FB_SetupCtrlHold;
	m_armManualAdjust :ARRAY[1..g_sArmNum] OF FB_SetupCtrlManualAdjust;
	m_armAutoAdjust :ARRAY[1..g_sArmNum] OF FB_SetupCtrlAutoAdjust;
	m_armPackage :ARRAY[1..g_sArmNum] OF FB_SetupCtrlPackage;
	m_armCart :ARRAY[1..g_sArmNum] OF FB_SetupCtrlCart;
	m_armJnt3GraCali :ARRAY[1..g_sArmNum] OF FB_SetupCtrlJnt3GraCali;
	m_armJnt5GraCali :ARRAY[1..g_sArmNum] OF FB_SetupCtrlJnt5GraCali;
	m_armDisable :ARRAY[1..g_sArmNum] OF FB_SetupCtrlDisable;
	
	
	// arm controller interface
	m_armCtrl :ARRAY[1..g_sArmNum] OF I_SetupArmCtrl;
	m_armCtrlCmds :ARRAY[1..g_sArmNum] OF ST_SetupArmCtrlCmds;

END_VAR

METHOD PUBLIC getStatus : BOOL
VAR_IN_OUT
	// slave robot information, including arm status and cartesian data
	r_setupStatus :ST_SetupStatus;
	
	// slave robot joint data
	r_setupJointsData :ST_SetupJointData;
	
END_VAR

VAR
	i:INT;
END_VAR
r_setupStatus.m_armState:=m_setupArmState;

// TODO: project cartesion data to monitor coordinate
FOR i:=1 TO g_sArmNum DO
	
	// cartesion
	r_setupStatus.m_curEndPose[i]:=m_setupArms[i].curCartPose;
	r_setupStatus.m_rcPos[i]:=m_setupArms[i].rcPos;
	
	// joint
	r_setupJointsData.m_curMotorPos[i]:=m_setupArms[i].curMotorPos;
	r_setupJointsData.m_curLinkPos[i]:=m_setupArms[i].curLinkPos;
	r_setupJointsData.m_curJntPos[i]:=m_setupArms[i].curJntPos;
	r_setupJointsData.m_curJntVel[i]:=m_setupArms[i].curJntVel;
	r_setupJointsData.m_curJntTrq[i]:=m_setupArms[i].curJntTrq;
	
	// command info
	// joint info
	r_setupJointsData.m_cmdJntPos[i]:=m_armCtrlCmds[i].m_cmdJntPos;
	r_setupJointsData.m_cmdJntVel[i]:=m_armCtrlCmds[i].m_cmdJntVel;
	r_setupJointsData.m_cmdJntTrq[i]:=m_armCtrlCmds[i].m_cmdJntTrq;
	
END_FOR
END_METHOD

METHOD PUBLIC Init : BOOL
VAR_INPUT
END_VAR
VAR
	i:INT;
END_VAR
FOR i:=1 TO g_sArmNum DO
	// arm init
	m_setupArms[i].Init(i);
	m_setupArmState[i]:=SlaveArmState_Init;
	m_lastSetupArmState[i]:=SlaveArmState_Init;
	m_nextSetupArmState[i]:=SlaveArmState_Init;
	
	// command init
	m_armCtrlCmds[i].m_jntEnableFlag := g_zeroVec5i;
	m_armCtrlCmds[i].m_jntOPMode := g_setupAllPosMode;
	m_armCtrlCmds[i].m_cmdJntPos := m_setupArms[i].curJntPos;
	m_armCtrlCmds[i].m_cmdJntVel := g_zeroVec5d;
	m_armCtrlCmds[i].m_cmdJntAcc := g_zeroVec5d;
	m_armCtrlCmds[i].m_cmdJntTrq := g_zeroVec5d;
	
	// generate controller factory
	m_armCtrlFactory[i,SetupArmState_Error] := m_armError[i];
	m_armCtrlFactory[i,SetupArmState_Init] := m_armInit[i];
	m_armCtrlFactory[i,SetupArmState_SelfCheck] := m_armSelfCheck[i];
	m_armCtrlFactory[i,SetupArmState_Hold] := m_armHold[i];
	m_armCtrlFactory[i,SetupArmState_ManualAdjust] := m_armManualAdjust[i];
	m_armCtrlFactory[i,SetupArmState_AutoAdjust] := m_armAutoAdjust[i];
	m_armCtrlFactory[i,SetupArmState_Package] := m_armPackage[i];
	m_armCtrlFactory[i,SetupArmState_Cart] := m_armCart[i];
	m_armCtrlFactory[i,SetupArmState_jnt3GravityCali] := m_armJnt3GraCali[i];
	m_armCtrlFactory[i,SetupArmState_jnt5GravityCali] := m_armJnt5GraCali[i];
	m_armCtrlFactory[i,SetupArmState_Disable] := m_armDisable[i];
	
	// assign controller
	m_armCtrl[i]:=m_armCtrlFactory[i,m_setupArmState[i]];
	m_armCtrl[i].Init(m_setupArms[i],m_armCtrlCmds[i]);
END_FOR
END_METHOD

METHOD PUBLIC run : BOOL
VAR_IN_OUT CONSTANT
	i_setupInputDataPool:ST_SetupInputDataPool;
END_VAR
VAR
	i:INT;
END_VAR
// state machine transition
stateMachine(i_setupInputDataPool);

FOR i:=1 TO g_sArmNum DO
	// update dynamic data
	m_setupArms[i].updateDyna(i_setupInputDataPool.m_setupJnt3Gravity[i], i_setupInputDataPool.m_setupJnt5Gravity[i]);
								
	// update slave arm kinematics
	m_setupArms[i].updateStatus();
	
	// null ptr check
	IF 0 = m_armCtrl[i] THEN
		EXIT;
	END_IF
	
	// run controller
	m_armCtrl[i].run(m_setupArms[i],m_armCtrlCmds[i]);

	// update commands to drivers
	m_setupArms[i].updateCmds(m_armCtrlCmds[i]);

END_FOR
END_METHOD

// state machine check and transit 
METHOD PROTECTED stateMachine : BOOL
VAR_IN_OUT CONSTANT
		i_setupInputDataPool:ST_SetupInputDataPool;
END_VAR
VAR
	i:INT;
END_VAR
FOR i:=1 TO g_sArmNum DO
	// State machine transit 
	CASE m_setupArmState[i] OF
		// error
		SetupArmState_Error:
			IF FALSE = i_setupInputDataPool.m_safetyData.m_setupErrFlag[i]  THEN
				m_nextSetupArmState[i]:=SetupArmState_Hold;
			END_IF
			
		// init
		SetupArmState_Init:
			// to hold. No self check for setup arm currently
			IF m_armCtrl[i].isFinished  THEN
				m_nextSetupArmState[i]:=SetupArmState_Hold;
			END_IF

		//self check
		SetupArmState_SelfCheck:
			IF m_armCtrl[i].isFinished  THEN
				m_nextSetupArmState[i]:=SetupArmState_Hold;
			END_IF
		
		//hold
		SetupArmState_Hold:
			// to manual adjust
			IF m_setupArms[i].manualAdjustOn OR m_setupArms[i].m_jnt5AdjustDir<>0 THEN
				m_nextSetupArmState[i]:=SetupArmState_ManualAdjust;
			END_IF
			
		
		// manual adjust
		SetupArmState_ManualAdjust:
			// to hold
			IF NOT(m_setupArms[i].manualAdjustOn) AND m_setupArms[i].jnt5AdjustDir=0 THEN
				m_nextSetupArmState[i] := SetupArmState_Hold;
			END_IF
			
		// auto adjust
		SetupArmState_AutoAdjust:
				
		//package
		SetupArmState_Package:
		
		//cart
		SetupArmState_Cart:
		
		//joint 5 gravity calibration
		SetupArmState_jnt5GravityCali:
			IF m_armCtrl[i].isFinished  THEN
				m_nextSetupArmState[i]:=SetupArmState_Hold;
			END_IF 
			
		//joint 3 gravity calibration
		SetupArmState_jnt3GravityCali:
			IF m_armCtrl[i].isFinished  THEN
				m_nextSetupArmState[i]:=SetupArmState_Hold;
			END_IF 
		
		// arm disable
		SetupArmState_Disable:
			IF NOT(i_setupInputDataPool.m_UIData.m_slaveArmDisableFlag[i]) THEN
				m_nextSetupArmState[i]:= SetupArmState_Hold;
			END_IF
	END_CASE
	
	// arm disable
	IF i_setupInputDataPool.m_UIData.m_slaveArmDisableFlag[i] AND m_setupArmState[i] <> SetupArmState_Init THEN
		m_nextSetupArmState[i] := SetupArmState_Disable;
	// error check
	ELSIF i_setupInputDataPool.m_safetyData.m_setupErrFlag[i] THEN
		m_nextSetupArmState[i]:=SetupArmState_Error;
	END_IF
	
	// Controller transit
	IF m_nextSetupArmState[i]<> m_setupArmState[i] THEN
		// reset current controller
		m_armCtrl[i].reset();
		
		// transit to new controller
		m_lastSetupArmState[i]:=m_setupArmState[i];
		m_setupArmState[i]:=m_nextSetupArmState[i];
		m_armCtrl[i]:=m_armCtrlFactory[i,m_setupArmState[i]];
		
		// init next controller
		m_armCtrl[i].Init(m_setupArms[i],m_armCtrlCmds[i]);
		m_setupArms[i].updateCmds(m_armCtrlCmds[i]);
	END_IF
END_FOR
END_METHOD

END_FUNCTION_BLOCK

// ---- FBs_SetupControllers/FB_SetupCtrlJnt3GraCali.TcPOU
// Brief: setup arm gravity calibration
// For trajectory synchronizaiton, the planner generate a trajecotry for setup joint3/5 and slave joint 1-3, but only former used here 
FUNCTION_BLOCK PUBLIC FB_SetupCtrlJnt3GraCali EXTENDS FB_SetupArmCtrlBase
VAR_INPUT
END_VAR
VAR_OUTPUT
END_VAR
VAR
// cali trajectory
	m_caliMotionSegs :INT :=3;
	m_graCaliTraj:ARRAY [1..3] OF LREAL:=[0.002,0.198,0.002];
	
	m_caliMaxjntVel:LREAL:=0.01;
	m_caliMaxjntAcc:LREAL:=0.5;
	m_caliMaxjntJerk:LREAL:=1.0;
	
	m_caliTrajIdx: INT := 1;
	m_caliPlanner: ARRAY[1..3] OF FB_BasicDoubleS;
	
END_VAR

// override this function in each exact controller
METHOD PROTECTED calcCmdJntPos : BOOL
VAR_IN_OUT CONSTANT
	i_setupArm	:FB_SetupArm;
END_VAR


VAR 
	i :INT;
	curJntVel :Vec5d;
END_VAR
// safety check
IF ABS(i_setupArm.curJntVel[3]) > 0.05 THEN
	m_isFinished:=TRUE;
	RETURN;
END_IF

// check if planner is ready
IF m_caliPlanner[m_caliTrajIdx].isGene = FALSE THEN
	calcCmdJntPos:=FALSE;
	RETURN;
END_IF

// traj plan
calcCmdJntPos :=m_caliPlanner[m_caliTrajIdx].evaluate(m_timePeriod, q=> m_cmdJntPos[3], q_dot=>m_cmdJntVel[3], q_ddot=> m_cmdJntAcc[3]);

// check if to transit to next segment
IF(m_timePeriod > m_caliPlanner[m_caliTrajIdx].duration  AND ABS(i_setupArm.curJntVel[3])<GVL_SlaveControlParameters.g_jntStaticVelThres) THEN
	m_caliTrajIdx:=m_caliTrajIdx+1;
	m_timePeriod:=0;
END_IF

// check if to terminated
IF(m_caliTrajIdx > m_caliMotionSegs) THEN
	m_isFinished:=TRUE;
END_IF
END_METHOD

METHOD PUBLIC init : BOOL
VAR_IN_OUT CONSTANT
	i_setupArm	:FB_SetupArm;
END_VAR
VAR_IN_OUT 
	r_setupArmCtrlCmd :ST_SetupArmCtrlCmds;
END_VAR

VAR
	i,j :INT;
	startJntPos,endJntPos :LREAL;
	q,v:ARRAY[1..2] OF lreal;
END_VAR
SUPER^.Init(i_setupArm,r_setupArmCtrlCmd);
m_jntEnableFlag[3]:=1;
m_jntOPMode[3]:= DriverOPMode_Pos;
m_caliTrajIdx :=1;

// traj plan
// fisrt segment
q[1]:=i_setupArm.curJntPos[3];
q[2]:=m_graCaliTraj[1];
v[1]:=0;
v[2]:=0;
m_caliPlanner[1].init(q,v,m_caliMaxjntVel, m_caliMaxJntAcc, m_caliMaxJntJerk);

// other segments
FOR i:=2 TO m_caliMotionSegs DO 
	q[1]:=m_graCaliTraj[i-1];
	q[2]:=m_graCaliTraj[i];
	m_caliPlanner[i].init(q,v,m_caliMaxjntVel, m_caliMaxJntAcc, m_caliMaxJntJerk);
END_FOR
END_METHOD

END_FUNCTION_BLOCK

// ---- FBs_SlaveControllers/FB_SlaveCtrlDisable.TcPOU
// Brief: Slave Arm Error Hold
FUNCTION_BLOCK PUBLIC FB_SlaveCtrlDisable EXTENDS FB_SlaveArmCtrlBase
VAR_INPUT
END_VAR
VAR_OUTPUT
END_VAR
VAR
END_VAR

// override this function in each exact controller
METHOD PROTECTED calcCmdJntPos : BOOL
VAR_IN_OUT CONSTANT
	// endoscope pose in cart coordinate
	i_endoscopePose : ST_Frame;
	
	// master arm data
	i_masterStatus :ST_MasterStatus;
	
	// setup arm data
	i_setupStatus: ST_SetupStatus;
	
	// slave arm data
	i_slaveArm :FB_SlaveArm;
END_VAR
m_cmdJntPos := i_slaveArm.curJntPos;
END_METHOD

// override this function in each exact controller
// NOTICE: set joint control mode here, and do some initialization if needed
METHOD PUBLIC init : BOOL
VAR_IN_OUT CONSTANT
	i_slaveArm	:FB_SlaveArm;
END_VAR
VAR_IN_OUT 
	r_slaveArmCtrlCmd :ST_SlaveArmCtrlCmds;
END_VAR


VAR
	i:INT;
END_VAR
SUPER^.Init(i_slaveArm,r_slaveArmCtrlCmd);

// disable all joints
 m_jntEnableFlag :=g_zeroVec8i;
 
 // update commands to arm
copyCmds(r_slaveArmCtrlCmd);
END_METHOD

END_FUNCTION_BLOCK

// ---- FBs_SlaveControllers/FB_SlaveCtrlInstruReady.TcPOU
// Brief: Instrument Ready
FUNCTION_BLOCK PUBLIC FB_SlaveCtrlInstruReady EXTENDS FB_SlaveArmCtrlBase
VAR_INPUT
END_VAR
VAR_OUTPUT
END_VAR
VAR
END_VAR

METHOD PUBLIC init : BOOL
VAR_IN_OUT CONSTANT
	i_slaveArm	:FB_SlaveArm;
END_VAR
VAR_IN_OUT 
	r_slaveArmCtrlCmd :ST_SlaveArmCtrlCmds;
END_VAR


VAR
	j:INT;
	maxJntErr:LREAL;
	jntCtrlErr:Vec7d;
END_VAR
// DO NOT hold last command
//m_holdLastCmds := checkToHoldLastCmds(i_slaveArm);

//init
SUPER^.Init(i_slaveArm,r_slaveArmCtrlCmd);
END_METHOD

END_FUNCTION_BLOCK

// ---- FBs_SlaveControllers/FB_SlaveCtrlMasterSlave.TcPOU
// Brief: Slave Arm MasterSlave controller
FUNCTION_BLOCK PUBLIC FB_SlaveCtrlMasterSlave EXTENDS FB_SlaveArmCtrlBase
VAR_INPUT
END_VAR
VAR_OUTPUT
END_VAR
VAR
	// master-slave motion scale
	m_MSMotionScale :LREAL;
		
	// gripper match angle threshold
	m_gripperMatchAngThres :LREAL := 2*g_deg2Rad;
	
	// control error thershold for safety check
	m_maxPosTrackErr :LREAL := 0.05;
	m_maxOriTrackErr :LREAL :=g_deg2Rad * 30;
	
	// filter cut-off frequency for master-slave control
	m_cmdJntPosLpfCutoffFreq : LREAL :=5;
	
	// last command joint position
	m_lastCmdJntPos :Vec8d;
	
	// simulated DH joint position
	m_simDHJntPos : Vec6d;
	
	// simulated slave twist of DH joint
	m_simDHJointVel :Vec6d;
		
	// enter master-slave control for the first time
	m_firstIn :BOOL := TRUE;
	
	// flag if reach joint limit
	m_reachMacroJntLimit :BOOL;
	m_reachWristJntLimit :BOOL;
	
	// master/slave origin pose when first enter master-slave control
	m_masterOriginPose : ST_Frame;
	m_slaveOriginPose : ST_Frame;
	
	// orientation deviation(in master coordinate) between master and slave when first enter control
	m_MSOriDeviation : Mat3d;
	
	// command joint position filter
	m_cmdJntPosLpf:ARRAY[1..8] OF FB_LowPassFilter;
	
	// commmand yaw angle and velocity
	m_cmdYawAngle :LREAL;
	m_cmdYawVel :LREAL;
	
	// comand yaw angle and velocity filter
	m_cmdYawAngLpf : FB_LowPassFilter;
	m_cmdYawVelLpf : FB_LowPassFilter;
	
	// master pose/velocity in monitor coordinate
	m_masterPose :ST_Frame;
	m_masterTwist : Vec6d;
	
	// master grip angle
	m_masterGripAngle : LREAL;
	
	// slave command/current pose in endoscope coordinate
	m_slaveCmdPoseInScope :ST_Frame;
	m_slavePoseInScope : ST_Frame;
	
	// slave command/current pose in cart
	m_slaveCmdPoseInCart :ST_Frame;
	m_slavePoseInCart : ST_Frame;
	
	// instrument controller
	m_instruController : FB_InstrumentControl;
	
	// slave command grip angle and grip force level
	m_slaveCmdGripAngle :LREAL;
	m_slaveCmdGripForceLevel:LREAL;
	
	// slave pose error
	m_slavePosErr :Vec3d;
	m_slaveRotErr :Mat3d;
	m_errAngle : LREAL;
	m_errAxisLocal, m_errAxis :Vec3d;
	m_masterSlavePoseError :Vec6d;
	
	// velocity for slave to track master motion
	m_slaveTrackTwist :Vec6d;
	m_slaveCmdVel, m_slaveCmdWVel : Vec3d;
	
	// last master gripper angle
	m_lastMasterGripAngle :LREAL;
	
	// master gripper angle velocity
	m_masterGripAngleVel :LREAL;
	m_masterGripAngleVelLpf :FB_LowPassFilter;
	
	// flag to start gripper control
	m_gripperCtrlFlag :BOOL;
	
	// code execute time measure
	m_codeTime : Profiler;
	
END_VAR

METHOD PROTECTED calcCmdJntPos : BOOL
VAR_IN_OUT CONSTANT
	i_endoscopePose : ST_Frame;
	i_masterStatus :ST_MasterStatus;
	i_setupStatus: ST_SetupStatus;
	i_slaveArm :FB_SlaveArm;
END_VAR

VAR 
	i,j : INT;
	tmpMat3d : Mat3d;
	masterMotionRange : Vec3d;
	
	masterVelInScope, masterWVelInScope :Vec3d;
	masterVelInCart, masterWVelInCart :Vec3d;

	cmdVelScale :LREAL;
	invJaco :Mat6d;
	DHJntCmdDeltaPos :Vec6d;
	armJntJaco,armJntJacoInv, wristJntJaco :Mat3d;
	velByWristJnt,velByArmJnt : Vec3d;
	armDHJntVel, wristDHJntVel :Vec3d;
	tmpFrame : ST_Frame;
	slaveSimDHJntPos :Vec6d;
	
END_VAR
m_codeTime(START:=TRUE, RESET:=TRUE);

IF isFinished THEN
	RETURN;
END_IF

// decide matched master arm index
FOR i:=1 TO g_mArmNum DO 
	IF i_masterStatus.m_teleSlaveArmIdx[i] = i_slaveArm.armIdx THEN
		m_masterPose := i_masterStatus.m_curArmPose[i];
		m_masterTwist := i_masterStatus.m_curArmTwist[i];
		m_masterGripAngle := i_masterStatus.m_gripAngle[i];
	END_IF
END_FOR

// compute slave pose in endoscope coordinate
m_slavePoseInCart := transform(i_setupStatus.m_curEndPose[i_slaveArm.armIdx], i_slaveArm.simCartPose);
tmpFrame :=invFrame(i_endoscopePose);
m_slavePoseInScope := transform(tmpFrame, m_slavePoseInCart);

// handle for the first time in
IF TRUE = m_firstIn THEN
	m_firstIn := FALSE;
	m_masterOriginPose :=m_masterPose;
	m_slaveOriginPose := m_slavePoseInScope;
	matTranspose(m_masterOriginPose.m_rot, tmpMat3d);
	matMultiply(tmpMat3d, m_slavePoseInScope.m_rot,m_MSOriDeviation);
	m_lastMasterGripAngle := m_masterGripAngle;
	
	// only update motion scale while entering teleControl 
	m_MSMotionScale := 1.0/ MAX(1,  i_masterStatus.m_motionScale);
END_IF

// compute master twist in slave arm coordinate
(*FOR i:=1 TO 3 DO
	masterVelInScope[i] := m_masterTwist[i]*i_masterStatus.m_motionScale;
	masterWVelInScope[i] := m_masterTwist[i+3];
END_FOR
matMultiVec(i_endoScopePose.m_rot, masterVelInScope, masterVelInCart);
matMultiVec(i_endoScopePose.m_rot, masterWVelInScope, masterWVelInCart);
matTranspose(i_setupStatus.m_curEndPose[i_slaveArm.armIdx].m_rot, tmpMat3d);
matMultiVec(tmpMat3d,masterVelInCart, m_masterFFVel);
matMultiVec(tmpMat3d,masterWVelInCart, m_masterFFWVel);
FOR i:=1 TO 3 DO
	m_cmdCartTwist[i] := m_masterFFVel[i];
	m_cmdCartTwist[i+3] := m_masterFFWVel[i];
END_FOR*)

// compute slave command pose in scope
vecSub(m_masterPose.m_pos, m_masterOriginPose.m_pos, masterMotionRange);

vecSelfMultiNum(masterMotionRange, m_MSMotionScale);
vecAdd(m_slaveOriginPose.m_pos, masterMotionRange, m_slaveCmdPoseInScope.m_pos);
matMultiply(m_masterPose.m_rot, m_MSOriDeviation, m_slaveCmdPoseInScope.m_rot);

// compute slave command pose in slave arm coordinate
m_slaveCmdPoseInCart := transform(i_endoScopePose, m_slaveCmdPoseInScope);
tmpFrame := invFrame(i_setupStatus.m_curEndPose[i_slaveArm.armIdx]);
m_cmdCartPose := transform(tmpFrame, m_slaveCmdPoseInCart);

// compute pose error
vecSub(m_cmdCartPose.m_pos, i_slaveArm.simCartPose.m_pos, m_slavePosErr);

matTranspose(i_slaveArm.simCartPose.m_rot, tmpMat3d);
matMultiply(tmpMat3d, m_cmdCartPose.m_rot, m_slaveRotErr);
rot2AngAxis(m_slaveRotErr, angle=>m_errAngle, axis=>m_errAxisLocal);
matMultiVec(i_slaveArm.simCartPose.m_rot, m_errAxisLocal, m_errAxis);

// calculate pose error in endoscope
calcMSErrInScope(i_endoscopePose, i_setupStatus.m_curEndPose[i_slaveArm.armIdx]);

// safety check
(*IF norm(m_slavePosErr) > m_maxPosTrackErr OR ABS(m_errAngle)>m_maxOriTrackErr THEN
	m_isFinished := TRUE;
END_IF*) 

// pose track control
vecMultiNum(m_slavePosErr, g_slaveArmCtrlFreq, m_slaveCmdVel);
vecMultiNum(m_errAxis, m_errAngle*g_slaveArmCtrlFreq, m_slaveCmdWVel);
FOR i:=1 TO 3 DO 
	m_slaveTrackTwist[i] := m_slaveCmdVel[i];
	m_slaveTrackTwist[i+3] := m_slaveCmdWVel[i];
END_FOR

// compute command velocity for DH joints
invJaco := i_slaveArm.simJacoInv;
matMultiVec(invJaco, m_slaveTrackTwist, m_simDHJointVel);

// limit DH joints velocity 
cmdVelScale := 1;
FOR i:=1 TO g_cartDofs DO 
	cmdVelScale:=MAX(cmdVelScale, ABS(m_simDHJointVel[i]/GVL_SlaveMotorParameters.g_maxJntVel[i]));
END_FOR
vecSelfMultiNum(m_simDHJointVel, 1.0/cmdVelScale);
vecSelfMultiNum(m_slaveTrackTwist, 1.0/cmdVelScale);
vecSelfMultiNum(m_slaveCmdVel, 1.0/cmdVelScale);
vecSelfMultiNum(m_slaveCmdWVel, 1.0/cmdVelScale);

// limit instrument wrist joint position
FOR i:=1 TO 3 DO
	armDHJntVel[i]:=m_simDHJointVel[i];
	wristDHJntVel[i]:=m_simDHJointVel[i+3];
END_FOR

m_reachWristJntLimit :=FALSE;
FOR i:=1 TO 3 DO
	IF (wristDHJntVel[i] > 0 AND i_slaveArm.simDHJntPos[i+3] + wristDHJntVel[i]*g_slaveArmCtrlCycleTime> GVL_SlaveMotorParameters.g_maxDHJntPos[i+3]) OR 
		(wristDHJntVel[i]<0 AND i_slaveArm.simDHJntPos[i+3] + wristDHJntVel[i]*g_slaveArmCtrlCycleTime< GVL_SlaveMotorParameters.g_minDHJntPos[i+3]) OR
		ABS(m_errAngle)>m_maxOriTrackErr THEN
		wristDHJntVel:=g_zeroVec3d;
		m_reachWristJntLimit:=TRUE;
		CONTINUE;
	END_IF
END_FOR

// modify arm joints velocity to compensate wrist joint motion
FOR i:=1 TO 3 DO
	FOR j:=1 TO 3 DO
		armJntJaco[i,j]:=i_slaveArm.simJaco[i,j];
		wristJntJaco[i,j]:=i_slaveArm.simJaco[i,j+3];
	END_FOR
END_FOR
invMat3(armJntJaco, armJntJacoInv);
matMultiVec(wristJntJaco, wristDHJntVel, velByWristJnt);
vecSub(m_slaveCmdVel, velByWristJnt, velByArmJnt);
matMultiVec(armJntJacoInv, velByArmJnt, armDHJntVel);

// limit DH joints velocity 
cmdVelScale := 1;
FOR i:=1 TO 3 DO 
	cmdVelScale:=MAX(cmdVelScale, ABS(armDHJntVel[i]/GVL_SlaveMotorParameters.g_maxJntVel[i]));
END_FOR
vecSelfMultiNum(armDHJntVel, 1.0/cmdVelScale);

// limit arm joint position
m_reachMacroJntLimit :=FALSE;
FOR i:=1 TO 3 DO
	IF (armDHJntVel[i] > 0 AND  i_slaveArm.simDHJntPos[i] + armDHJntVel[i]*g_slaveArmCtrlCycleTime> GVL_SlaveMotorParameters.g_maxDHJntPos[i]) OR 
		(armDHJntVel[i] <0 and	i_slaveArm.simDHJntPos[i] + armDHJntVel[i]*g_slaveArmCtrlCycleTime< GVL_SlaveMotorParameters.g_minDHJntPos[i]) THEN
		armDHJntVel[i]:=0;
		m_reachMacroJntLimit:=TRUE;
	END_IF
END_FOR

// integrate command DH joint position
FOR i:=1 TO 3 DO
	m_simDHJointVel[i]:=armDHJntVel[i];
	m_simDHJointVel[i+3]:=wristDHJntVel[i];
END_FOR
vecMultiNum(m_simDHJointVel, g_slaveArmCtrlCycleTime, DHJntCmdDeltaPos);
slaveSimDHJntPos:=i_slaveArm.simDHJntPos;
vecAdd(slaveSimDHJntPos, DHJntCmdDeltaPos, m_simDHJntPos);

// gripper angle/force control
gripperControl(i_slaveArm);

// calculate target motor joint position/velocity from DH joint position
//i_slaveArm.instrument.gripAngleMap(m_masterGripAngle,o_instruGripAngle=>m_slaveCmdGripAngle, o_instruGripForceLevel=>m_slaveCmdGripForceLevel);
i_slaveArm.instrument.instruIK(m_simDHJntPos,m_slaveCmdGripAngle, o_jntPos=>m_simJntPos);

// filt command joint position
FOR i:=1 TO g_sJntNum DO 
	m_cmdJntPos[i] := m_cmdJntPosLpf[i].run(m_simJntPos[i]);
END_FOR

// compute command joint velocity
vecSub(m_cmdJntPos, m_lastCmdJntPos, m_cmdJntVel);
vecSelfMultiNum(m_cmdJntVel, g_slaveArmCtrlFreq);
m_lastCmdJntPos:=m_cmdJntPos;

m_codeTime(START:=FALSE);
END_METHOD

// override this function in each exact controller
METHOD PROTECTED calcCmdJntTrq : BOOL
VAR_IN_OUT CONSTANT
	i_endoscopePose : ST_Frame;
	i_masterStatus :ST_MasterStatus;
	i_setupStatus: ST_SetupStatus;
	i_slaveArm :FB_SlaveArm;
END_VAR
VAR
	i :INT ;
	instruCmdGripAngle, instruCmdGripForceLevel :LREAL;
	instruCmdJntPos, instruCmdJntVel : Vec5d;	
	instruJntCtrlTrq :Vec5d;
END_VAR
IF isFinished THEN
	RETURN;
END_IF

// set joint torque to zero in default
m_cmdJntTrq := g_zeroVec8d;

// instrument joint control
FOR i:=1 TO 5 DO 
	instruCmdJntPos[i]:=m_cmdJntPos[i+3];
	instruCmdJntVel[i]:=m_cmdJntVel[i+3];
END_FOR
m_cmdYawAngle := m_cmdYawAngLpf.run(m_simDHJntPos[6]);
m_cmdYawVel := m_cmdYawVelLpf.run(m_simDHJointVel[6]);
m_instruController.run(instruCmdJntPos,instruCmdJntVel, m_cmdYawAngle, m_cmdYawVel, m_slaveCmdGripForceLevel, i_slaveArm, o_cmdJntTrq=>instruJntCtrlTrq);

FOR i:=1 TO 5 DO
	m_cmdJntTrq[i+3]:=instruJntCtrlTrq[i];
END_FOR
END_METHOD

METHOD calcMSErrInScope : BOOL
VAR_IN_OUT CONSTANT
	i_endoscopePose : ST_Frame;
	i_setupPose :ST_Frame;
END_VAR
VAR
	posErrInCart,oriErrInCart :Vec3d;
	invRot :Mat3d;
	posErrInScope,oriErrInScope :Vec3d;
	i:INT;
END_VAR
m_masterSlavePoseError := g_zeroVec6d;

// pose error in cart coordinate
matMultiVec(i_setupPose.m_rot, m_slavePosErr, posErrInCart);
matMultiVec(i_setupPose.m_rot, m_errAxis, oriErrInCart);
vecSelfMultiNum(oriErrInCart, m_errAngle);

// pose err in endoscope coordinate
matTranspose(i_endoscopePose.m_rot, invRot);
matMultiVec(invRot, posErrInCart, posErrInScope);
matMultiVec(invRot, oriErrInCart, oriErrInScope);

IF m_reachMacroJntLimit THEN
	FOR i:=1 TO 3 DO 
		m_masterSlavePoseError[i]:=posErrInScope[i];
	END_FOR
END_IF
IF m_reachWristJntLimit THEN
	FOR i:=1 TO 3 DO 
		m_masterSlavePoseError[i+3]:=oriErrInScope[i];
	END_FOR
END_IF
END_METHOD

METHOD gripperControl : BOOL
VAR_IN_OUT CONSTANT
	i_slaveArm :FB_SlaveArm;
END_VAR

VAR
	matchedSlaveGripAngle:LREAL;
	matchedSlaveGripForce:LREAL;
	masterGripVelThres :LREAL := 5.0 *g_deg2Rad;
END_VAR
// compute master grip veloicty
m_masterGripAngleVel:= (m_masterGripAngle - m_lastMasterGripAngle)/g_slaveArmCtrlCycleTime;
m_masterGripAngleVel := m_masterGripAngleVelLpf.run(m_masterGripAngleVel);
m_lastMasterGripAngle :=m_masterGripAngle;

// compute matched slave grip angle and force
i_slaveArm.instrument.gripAngleMap(m_masterGripAngle,o_instruGripAngle=>matchedSlaveGripAngle, o_instruGripForceLevel=>matchedSlaveGripForce);

IF m_gripperCtrlFlag THEN
	m_slaveCmdGripAngle := matchedSlaveGripAngle;
	m_slaveCmdGripForceLevel := matchedSlaveGripForce;
	RETURN;
ELSE
	//m_gripperCtrlFlag := (ABS(m_masterGripAngleVel) >masterGripVelThres) AND  (m_masterGripAngleVel * (matchedSlaveGripAngle-i_slaveArm.curGripAngle)>0);
	m_gripperCtrlFlag := ABS(matchedSlaveGripAngle-i_slaveArm.curGripAngle)<m_gripperMatchAngThres OR 
		(matchedSlaveGripAngle<=i_SlaveArm.instrument.kinematicParameters.m_minGripAngle and i_slaveArm.curGripAngle<=i_SlaveArm.instrument.kinematicParameters.m_minGripAngle);
END_IF
END_METHOD

METHOD PUBLIC init : BOOL
VAR_IN_OUT CONSTANT
	i_slaveArm	:FB_SlaveArm;
END_VAR
VAR_IN_OUT 
	r_slaveArmCtrlCmd :ST_SlaveArmCtrlCmds;
END_VAR
VAR 
	i :INT ;
END_VAR
SUPER^.Init(i_slaveArm,r_slaveArmCtrlCmd);
m_simJntPos :=m_cmdJntPos;
m_lastCmdJntPos :=m_cmdJntPos;
m_jntOPMode[1] := DriverOPMode_PosTrq;
m_jntOPMode[2] := DriverOPMode_PosTrq;
m_jntOPMode[3] := DriverOPMode_PosTrq;
m_jntOPMode[4] := DriverOPMode_Trq;
m_jntOPMode[5] := DriverOPMode_Trq;
m_jntOPMode[6] := DriverOPMode_Trq;
m_jntOPMode[7] := DriverOPMode_Trq;
m_jntOPMode[8] := DriverOPMode_Trq;
m_firstIn :=TRUE;
m_gripperCtrlFlag :=false;

// init gripper angle
m_slaveCmdGripAngle := i_slaveArm.curGripAngle;
m_slaveCmdGripForceLevel:=0;

// init filter
FOR i:=1 TO g_sJntNum DO
	m_cmdJntPosLpf[i].init(1, m_cmdJntPosLpfCutoffFreq, g_slaveArmCtrlFreq);
END_FOR
m_cmdYawAngLpf.init(1, m_cmdJntPosLpfCutoffFreq, g_slaveArmCtrlFreq);
m_cmdYawVelLpf.init(1, m_cmdJntPosLpfCutoffFreq, g_slaveArmCtrlFreq);
m_masterGripAngleVelLpf.init(1, m_cmdJntPosLpfCutoffFreq, g_slaveArmCtrlFreq);

// init controller
m_instruController.init(i_slaveArm);

// update commands to arm
copyCmds(r_slaveArmCtrlCmd);
END_METHOD

PROPERTY masterSlavePoseErr : REFERENCE to Vec6d
GET
masterSlavePoseErr REF= m_masterSlavePoseError;
END_GET
END_PROPERTY

END_FUNCTION_BLOCK

// ---- FBs_SlaveControllers/FB_SlaveCtrlPanelReady.TcPOU
// Brief: Panel Ready
FUNCTION_BLOCK PUBLIC FB_SlaveCtrlPanelReady EXTENDS FB_SlaveArmCtrlBase
VAR_INPUT
END_VAR
VAR_OUTPUT
END_VAR
VAR
END_VAR

END_FUNCTION_BLOCK

// ---- FBs_Robots/FB_SlaveRobot.TcPOU
FUNCTION_BLOCK FB_SlaveRobot
VAR_INPUT
END_VAR
VAR_OUTPUT
END_VAR
VAR
	// flag if robot self-check passed
	m_selfCheckPass :ARRAY[1..g_sArmNum] OF BOOL :=[4(false)];
	
	// flag if master are connected
	m_masterOnLine :BOOL :=FALSE;
	m_masterOnLineCheck :FB_masterConnectionCheck;
	
	// master-slave motion scale
	m_motionScale :LREAL;
	
	// index(0 to 4) of slave arm which is tele-linked to master arm
	m_teleSlaveArmIdx :ARRAY[1..g_mArmNum] OF E_MatchedSlaveArmIdx;
	
	// flag if endoscope is mounted
	m_endoscopeMounted :BOOL := FALSE;
	
	// endoscope pose in cart coordinate
	m_endoscopePose : ST_Frame;
	
	// slave arms, responsible for arm kinematic and control
	m_slaveArms :ARRAY[1..g_sArmNum] OF FB_SlaveArm;
	
	// arm state
	m_slaveArmState:ARRAY[1..g_sArmNum] OF E_SlaveArmState:=[4(E_SlaveArmState.SlaveArmState_Error)];
	m_lastSlaveArmState:ARRAY[1..g_sArmNum] OF E_SlaveArmState:=[4(E_SlaveArmState.SlaveArmState_Error)];
	m_nextSlaveArmState:ARRAY[1..g_sArmNum] OF E_SlaveArmState:=[4(E_SlaveArmState.SlaveArmState_Error)];
	
	// matched master arm state
	m_matchedMasterArmState :ARRAY[1..g_sArmNum] OF E_MasterArmState:=[4(E_MasterArmState.MasterArmState_Error)];
	
	// flag if panel and instrument mounted
	m_panelMountedFlag :ARRAY[1..g_sArmNum] OF BOOL :=[4(FALSE)];
	m_instrumentMountedFlag :ARRAY[1..g_sArmNum] OF BOOL :=[4(FALSE)];
	
	// flag if enable instrument invasion after it mounted
	m_instruInvasionEnableFlag :ARRAY[1..g_sArmNum] OF BOOL :=[4(FALSE)];
	
	// all arm controller instance 
	m_armCtrlFactory :ARRAY[1..g_sArmNum,1..SlaveArmState_totalNum] OF I_SlaveArmCtrl;
	m_armError :ARRAY[1..g_sArmNum] OF FB_SlaveCtrlError;
	m_armInit :ARRAY[1..g_sArmNum] OF FB_SlaveCtrlInit;
	m_armSelfCheck :ARRAY[1..g_sArmNum] OF FB_SlaveCtrlSelfCheck;
	m_armStandBy :ARRAY[1..g_sArmNum] OF FB_SlaveCtrlStandBy;
	m_mountPanel :ARRAY[1..g_sArmNum] OF FB_SlaveCtrlMountPanel;
	m_panelReady :ARRAY[1..g_sArmNum] OF FB_SlaveCtrlPanelReady;
	m_mountInstru :ARRAY[1..g_sArmNum] OF FB_SlaveCtrlMountInstru;
	m_instruReady :ARRAY[1..g_sArmNum] OF FB_SlaveCtrlInstruReady;
	m_armMasterSlave :ARRAY[1..g_sArmNum] OF FB_SlaveCtrlMasterSlave;
	m_scopeReady :ARRAY[1..g_sArmNum] OF FB_SlaveCtrlScopeReady;
	m_armEndoscope :ARRAY[1..g_sArmNum] OF FB_SlaveCtrlEndoscope;
	m_armAdjust :ARRAY[1..g_sArmNum] OF FB_SlaveCtrlAdjust;
	m_armPackage :ARRAY[1..g_sArmNum] OF FB_SlaveCtrlPackage;
	m_armCart :ARRAY[1..g_sArmNum] OF FB_SlaveCtrlCart;
	m_armGraCali :ARRAY[1..g_sArmNum] OF FB_SlaveCtrlGraCali;
	m_armTest :ARRAY[1..g_sArmNum] OF FB_SlaveCtrlTest;
	m_instruRetract :ARRAY[1..g_sArmNum] OF FB_SlaveCtrlInstruRetract;
	m_instruInvasion :ARRAY[1..g_sArmNum] OF FB_SlaveCtrlInstruInvasion;
	m_armDisable :ARRAY[1..g_sArmNum] OF FB_SlaveCtrlDisable;
	
	// arm controller interface
	m_armCtrl :ARRAY[1..g_sArmNum] OF I_SlaveArmCtrl;
	m_armCtrlCmds :ARRAY[1..g_sArmNum] OF ST_SlaveArmCtrlCmds;

END_VAR

METHOD PROTECTED controllerTransit : BOOL
VAR_INPUT
END_VAR
VAR
	i:int;
END_VAR
FOR i:=1 TO g_sArmNum DO 
	// Controller transit
	IF m_nextSlaveArmState[i]<> m_slaveArmState[i] THEN
		// reset current controller
		m_armCtrl[i].reset();
		
		// transit to new controller
		m_lastSlaveArmState[i]:=m_slaveArmState[i];
		m_slaveArmState[i]:=m_nextSlaveArmState[i];
		m_armCtrl[i]:=m_armCtrlFactory[i,m_slaveArmState[i]];
		
		// init next controller
		m_armCtrl[i].Init(m_slaveArms[i],m_armCtrlCmds[i]);
		m_slaveArms[i].updateCmds(m_armCtrlCmds[i]);
	END_IF
END_FOR
END_METHOD

METHOD PUBLIC getStatus : BOOL
VAR_IN_OUT
	// slave robot information, including arm status and cartesian data
	r_slaveStatus :ST_SlaveStatus;
	
	// slave robot joint data
	r_slaveJointsData :ST_SlaveJointData;
	
END_VAR

VAR
	i:INT;
END_VAR
r_slaveStatus.m_armState:=m_slaveArmState;
r_slaveStatus.m_endoscopeMounted :=m_endoscopeMounted;
r_slaveStatus.m_endoscopePose :=m_endoscopePose;

FOR i:=1 TO g_sArmNum DO
	r_slaveStatus.m_selfCheckPass[i] := m_selfCheckPass[i];	

	// instrument data
	r_slaveStatus.m_instruStauts[i].m_type:=m_slaveArms[i].instrument.onChipData.m_Instrutype;
	r_slaveStatus.m_instruStauts[i].m_ready:=m_instrumentMountedFlag[i];
	r_slaveStatus.m_instruStauts[i].m_fingerAngle:=m_slaveArms[i].curGripAngle;
	
	// cartesion
	r_slaveStatus.m_curArmPose[i]:=m_slaveArms[i].curCartPose;
	r_slaveStatus.m_curArmTwist[i]:=m_slaveArms[i].curCartTwist;
	r_slaveStatus.m_masterSlavePoseError[i] := m_armMasterSlave[i].masterSlavePoseErr;
	// joint
	r_slaveJointsData.m_curMotorPos[i]:=m_slaveArms[i].curMotorPos;
	r_slaveJointsData.m_curLinkPos[i]:=m_slaveArms[i].curLinkPos;
	r_slaveJointsData.m_curJntPos[i]:=m_slaveArms[i].curJntPos;
	r_slaveJointsData.m_curJntVel[i]:=m_slaveArms[i].curJntVel;
	r_slaveJointsData.m_curJntTrq[i]:=m_slaveArms[i].curJntTrq;
	
	// command info
	// cartesion
	r_slaveStatus.m_cmdArmPose[i]:=m_slaveArms[i].cmdCartPose;
	r_slaveStatus.m_cmdArmTwist[i]:=m_slaveArms[i].cmdCartTwist;
	// joint info
	r_slaveJointsData.m_cmdJntPos[i]:=m_slaveArms[i].cmdJntPos;
	r_slaveJointsData.m_cmdJntVel[i]:=m_slaveArms[i].cmdJntVel;
	r_slaveJointsData.m_cmdJntTrq[i]:=m_slaveArms[i].cmdJntTrq;
	
END_FOR
END_METHOD

METHOD PUBLIC Init : BOOL
VAR_INPUT
END_VAR
VAR
	i:INT;
END_VAR
FOR i:=1 TO g_sArmNum DO
	// arm init
	m_slaveArms[i].Init(i);
	m_slaveArmState[i]:=SlaveArmState_Init;
	m_lastSlaveArmState[i]:=SlaveArmState_Init;
	m_nextSlaveArmState[i]:=SlaveArmState_Init;
	m_selfCheckPass[i]:=false;
	
	// command init
	m_armCtrlCmds[i].m_jntEnableFlag := g_zeroVec8i;
	m_armCtrlCmds[i].m_jntOPMode := g_slaveAllPosMode;
	m_armCtrlCmds[i].m_cmdCartPose := m_slaveArms[i].curCartPose;
	m_armCtrlCmds[i].m_cmdCartTwist := g_zeroVec6d;
	m_armCtrlCmds[i].m_cmdJntPos := m_slaveArms[i].curJntPos;
	m_armCtrlCmds[i].m_cmdJntVel := g_zeroVec8d;
	m_armCtrlCmds[i].m_cmdJntAcc := g_zeroVec8d;
	m_armCtrlCmds[i].m_cmdJntTrq := g_zeroVec8d;
	
	// generate controller factory
	m_armCtrlFactory[i,SlaveArmState_Error] := m_armError[i];
	m_armCtrlFactory[i,SlaveArmState_Init] := m_armInit[i];
	m_armCtrlFactory[i,SlaveArmState_SelfCheck] := m_armSelfCheck[i];
	m_armCtrlFactory[i,SlaveArmState_Standby] := m_armStandBy[i];
	m_armCtrlFactory[i,SlaveArmState_MountPanel] := m_mountPanel[i];
	m_armCtrlFactory[i,SlaveArmState_PanelReady] := m_panelReady[i];
	m_armCtrlFactory[i,SlaveArmState_MountInstru] := m_mountInstru[i];
	m_armCtrlFactory[i,SlaveArmState_InstruReady] := m_instruReady[i];
	m_armCtrlFactory[i,SlaveArmState_MasterSlave] := m_armMasterSlave[i];
	m_armCtrlFactory[i,SlaveArmState_ScopeReady] := m_scopeReady[i];
	m_armCtrlFactory[i,SlaveArmState_EndoScope] := m_armEndoscope[i];
	m_armCtrlFactory[i,SlaveArmState_Adjust] := m_armAdjust[i];
	m_armCtrlFactory[i,SlaveArmState_Package] := m_armPackage[i];
	m_armCtrlFactory[i,SlaveArmState_Cart] := m_armCart[i];
	m_armCtrlFactory[i,SlaveArmState_GravityCali] := m_armGraCali[i];
	m_armCtrlFactory[i,SlaveArmState_Test] := m_armTest[i];
	m_armCtrlFactory[i,SlaveArmState_InstruRetract] := m_instruRetract[i];
	m_armCtrlFactory[i,SlaveArmState_InstruInvasion] := m_instruInvasion[i];
	m_armCtrlFactory[i,SlaveArmState_Disable] := m_armDisable[i];
	
	// assign controller
	m_armCtrl[i]:=m_armCtrlFactory[i,m_slaveArmState[i]];
	m_armCtrl[i].Init(m_slaveArms[i],m_armCtrlCmds[i]);
END_FOR
END_METHOD

METHOD PUBLIC run : BOOL
VAR_IN_OUT CONSTANT
	i_slaveInputDataPool:ST_SlaveInputDataPool;
END_VAR
VAR
	i:INT;
END_VAR
m_motionScale := i_slaveInputDataPool.m_masterStatus.m_motionScale;
m_teleSlaveArmIdx := i_slaveInputDataPool.m_masterStatus.m_teleSlaveArmIdx;

// check master connection
m_masterOnLine := m_masterOnLineCheck.check(i_slaveInputDataPool.m_masterStatus.m_masterHeartBeat);

// check if endoscope is mounted
m_endoscopeMounted := FALSE;
FOR i:=1 TO g_sArmNum DO 
	IF m_slaveArms[i].instrument.onChipData.m_Instrutype=InstruType_endoscope THEN
		m_endoscopeMounted := TRUE;
		m_endoscopePose := transform(i_slaveInputDataPool.m_setupStatus.m_curEndPose[i], m_slaveArms[i].curCartPose);
	END_IF
END_FOR

// state machine transition
stateMachine(i_slaveInputDataPool);

// controller transition
controllerTransit();

FOR i:=1 TO g_sArmNum DO
	// update dynamic data
	m_slaveArms[i].updateDyna(i_slaveInputDataPool.m_slaveDynaData);
								
	// update slave arm kinematics
	m_slaveArms[i].updateStatus();
	
	// null ptr check
	IF 0 = m_armCtrl[i] THEN
		EXIT;
	END_IF
	
	// run controller
	m_armCtrl[i].run(m_endoscopePose, i_slaveInputDataPool.m_MasterStatus,
					i_slaveInputDataPool.m_setupStatus, m_SlaveArms[i],m_armCtrlCmds[i]);

	// update commands to drivers
	m_slaveArms[i].updateCmds(m_armCtrlCmds[i]);

END_FOR
END_METHOD

// state machine check and transit 
METHOD PROTECTED stateMachine : BOOL
VAR_IN_OUT CONSTANT
		i_slavesInputDataPool:ST_SlaveInputDataPool;
END_VAR
VAR
	i,j:INT;
END_VAR
// check instrument state
FOR i:=1 TO g_sArmNum DO
	// statues check
	IF m_slaveArms[i].panelOn = FALSE THEN
		m_panelMountedFlag[i]:=FALSE;
	END_IF
	IF m_slaveArms[i].instruOn = FALSE THEN
		m_instrumentMountedFlag[i]:=FALSE;
	END_IF
END_FOR

// get matched master arm state
FOR i:=1 TO g_sArmNum DO 
	m_matchedMasterArmState[i]:=MasterArmState_Error;
	FOR j:=1 TO g_mArmNum DO 
		IF i = i_slavesInputDataPool.m_masterStatus.m_teleSlaveArmIdx[j] THEN
			m_matchedMasterArmState[i] := i_slavesInputDataPool.m_masterStatus.m_armState[j];
		END_IF
	END_FOR
END_FOR

// check if to enable instrument invasion 
FOR i:=1 TO g_sArmNum DO
	IF SlaveArmState_Adjust = m_slaveArmState[i] OR SlaveArmState_Cart = m_slaveArmState[i] THEN
		m_instruInvasionEnableFlag[i]:=FALSE;
	ELSIF SlaveArmState_InstruRetract = m_slaveArmState[i] THEN
		m_instruInvasionEnableFlag[i]:=TRUE;
	END_IF
END_FOR  

// state machine transit
FOR i:=1 TO g_sArmNum DO
	CASE m_slaveArmState[i] OF
		// error
		SlaveArmState_Error:
			IF FALSE = i_slavesInputDataPool.m_safetyData.m_slaveErrFlag[i] THEN
				// to standby
				IF m_selfCheckPass[i] THEN
					m_nextSlaveArmState[i] :=SlaveArmState_Standby;
				// to init
				ELSE
					m_nextSlaveArmState[i] :=SlaveArmState_Init;
				END_IF
			END_IF
			
		// init
		SlaveArmState_Init:
			m_selfCheckPass[i]:=FALSE;
			// to selfcheck
			IF m_armCtrl[i].isFinished AND i_slavesInputDataPool.m_masterStatus.m_slaveSelfCheckFlag  THEN
				m_nextSlaveArmState[i]:=SlaveArmState_SelfCheck;
			// to adjust
			ELSIF m_slaveArms[i].adjustOn THEN
				m_nextSlaveArmState[i]:=SlaveArmState_Adjust;
			END_IF

		//self check
		SlaveArmState_SelfCheck:
			// to standby
			IF m_armCtrl[i].isFinished  THEN
				m_nextSlaveArmState[i]:=SlaveArmState_Standby;
				m_selfCheckPass[i]:=TRUE;
			END_IF
		
		//standby
		SlaveArmState_Standby:
			// to mount panel
			IF m_slaveArms[i].panelOn THEN 
				IF m_panelMountedFlag[i] THEN
					m_nextSlaveArmState[i]:=SlaveArmState_PanelReady;
				ELSE
					m_nextSlaveArmState[i]:=SlaveArmState_MountPanel;
				END_IF
			// to adjust
			ELSIF m_slaveArms[i].adjustOn THEN
				m_nextSlaveArmState[i]:=SlaveArmState_Adjust;
			END_IF
		
		//mount panel
		SlaveArmState_MountPanel:
			// to panel ready
			IF m_armCtrl[i]. isFinished THEN
				m_nextSlaveArmState[i]:=SlaveArmState_PanelReady;
				m_panelMountedFlag[i] :=TRUE;
				
				// NOTICE: multiple cycles joints back to center during initialization
				// 			need to reset joints encoder data again
				m_slaveArms[i].initJntPos();
			// to standby
			ELSIF NOT(m_slaveArms[i].panelOn) THEN
				m_nextSlaveArmState[i]:=SlaveArmState_Standby;
			END_IF
		
		//panel ready
		SlaveArmState_PanelReady:
			// to adjust
			IF (m_slaveArms[i].adjustOn) THEN
				m_nextSlaveArmState[i]:=SlaveArmState_Adjust;
			// to stand by
			ELSIF NOT(m_slaveArms[i].panelOn) THEN
				m_nextSlaveArmState[i]:=SlaveArmState_Standby;
			ELSIF m_slaveArms[i].instruOn  THEN
				IF m_instrumentMountedFlag[i] THEN
					// to scope ready
					IF  InstruType_endoscope = m_slaveArms[i].instrument.onChipData.m_Instrutype THEN 
						m_nextSlaveArmState[i]:=SlaveArmState_ScopeReady;
					// to instrument ready
					ELSE
						m_nextSlaveArmState[i]:=SlaveArmState_InstruReady;
					END_IF
				// to mount instrument/endoscope
				ELSE
					m_nextSlaveArmState[i]:=SlaveArmState_MountInstru;
				END_IF
			END_IF
			
		//mount instrument
		SlaveArmState_MountInstru:
			// to panel ready
			IF NOT m_slaveArms[i].instruOn THEN
				m_nextSlaveArmState[i]:=SlaveArmState_PanelReady;
			ELSIF m_armCtrl[i].isFinished THEN
				m_instrumentMountedFlag[i] :=TRUE;
				// NOTICE: multiple cycles joints back to center during initialization
				// 			need to reset joints encoder data again
				m_slaveArms[i].initJntPos();
				
				// record current joint position as offset for instrument
				m_slaveArms[i].instrument.initInstruJntPos(m_slaveArms[i].curJntPos);
				// to instrument invasion
				IF m_instruInvasionEnableFlag[i] THEN
					m_nextSlaveArmState[i] := SlaveArmState_InstruInvasion;
				// to endoscope ready
				ELSIF InstruType_endoscope = m_slaveArms[i].instrument.onChipData.m_Instrutype THEN
					m_nextSlaveArmState[i]:=SlaveArmState_ScopeReady;
				// to instrument ready
				ELSE
					m_nextSlaveArmState[i]:=SlaveArmState_InstruReady;
				END_IF
				
			END_IF
		
		// instrument ready
		SlaveArmState_InstruReady:
			// to instrument retract
			IF NOT m_slaveArms[i].instruOn THEN
				m_nextSlaveArmState[i]:=SlaveArmState_InstruRetract;
				m_slaveArms[i].recordInstruDepth();
			// to Adjust
			ELSIF (m_slaveArms[i].adjustOn) THEN
				m_nextSlaveArmState[i]:=SlaveArmState_Adjust;
			// to master-slave
			ELSIF MasterArmState_MasterSlave = m_matchedMasterArmState[i] THEN
				m_nextSlaveArmState[i] := SlaveArmState_MasterSlave;
			END_IF
		
		//master slave control
		SlaveArmState_MasterSlave:
			// to Adjust
			IF (m_slaveArms[i].adjustOn) THEN
				m_nextSlaveArmState[i]:=SlaveArmState_Adjust;
			// to standby
			ELSIF MasterArmState_MasterSlave <> m_matchedMasterArmState[i] THEN
				m_nextSlaveArmState[i]:=SlaveArmState_Standby;
			// to instrument retract
			ELSIF  NOT(m_slaveArms[i].panelOn) OR NOT(m_slaveArms[i].instruOn) THEN
				m_nextSlaveArmState[i]:=SlaveArmState_InstruRetract;
				m_slaveArms[i].recordInstruDepth();
			END_IF
		
		//endoscope ready
		SlaveArmState_ScopeReady:
			// to instrument retract
			IF NOT m_slaveArms[i].instruOn THEN
				m_nextSlaveArmState[i]:=SlaveArmState_InstruRetract;
				m_slaveArms[i].recordInstruDepth();
			// to Adjust
			ELSIF (m_slaveArms[i].adjustOn) THEN
				m_nextSlaveArmState[i]:=SlaveArmState_Adjust;
			// to endoscope control
			ELSIF MasterArmState_Endoscope = i_slavesInputDataPool.m_masterStatus.m_armState[1] AND 
				  MasterArmState_Endoscope = i_slavesInputDataPool.m_masterStatus.m_armState[2] THEN
				m_nextSlaveArmState[i] := SlaveArmState_EndoScope;
			END_IF
		
		//endoscope control
		SlaveArmState_EndoScope:
			// to Adjust
			IF (m_slaveArms[i].adjustOn) THEN
				m_nextSlaveArmState[i]:=SlaveArmState_Adjust;
			// to standby
			ELSIF MasterArmState_Endoscope <> i_slavesInputDataPool.m_masterStatus.m_armState[1]
				OR MasterArmState_Endoscope <> i_slavesInputDataPool.m_masterStatus.m_armState[2] THEN
				m_nextSlaveArmState[i]:=SlaveArmState_Standby;
			// to instrument retract
			ELSIF  NOT(m_slaveArms[i].panelOn) OR NOT(m_slaveArms[i].instruOn) THEN
				m_nextSlaveArmState[i]:=SlaveArmState_InstruRetract;
				m_slaveArms[i].recordInstruDepth();
			END_IF
			
		//arm adjust
		SlaveArmState_Adjust:
			IF NOT(m_slaveArms[i].adjustOn) THEN
				// to standby
				IF m_selfCheckPass[i] THEN
					m_nextSlaveArmState[i] :=SlaveArmState_Standby;
				// to init
				ELSE
					m_nextSlaveArmState[i] :=SlaveArmState_Init;
				END_IF
			END_IF
		
		// package
		SlaveArmState_Package:
			// to Adjust
			IF (m_slaveArms[i].adjustOn) THEN
				m_nextSlaveArmState[i]:=SlaveArmState_Adjust;
			// to standby
			ELSIF m_armCtrl[i].isFinished THEN
				m_nextSlaveArmState[i]:=SlaveArmState_Standby;
			END_IF
			
		// Cart
		SlaveArmState_Cart:
			IF NOT(i_slavesInputDataPool.m_cartStatus.m_inMotion) THEN
				// to standby
				IF m_selfCheckPass[i] THEN
					m_nextSlaveArmState[i] :=SlaveArmState_Standby;
				// to init
				ELSE
					m_nextSlaveArmState[i] :=SlaveArmState_Init;
				END_IF
			END_IF
		
		// Gravity Calibration
		SlaveArmState_GravityCali:
			// to Adjust
			IF (m_slaveArms[i].adjustOn) THEN
				m_nextSlaveArmState[i]:=SlaveArmState_Adjust;
			// to standby
			ELSIF m_armCtrl[i].isFinished THEN
				m_nextSlaveArmState[i]:=SlaveArmState_Standby;
			END_IF
			
		//arm test
		SlaveArmState_Test:
			// to standby
			IF  m_armCtrl[i].isFinished THEN
				m_nextSlaveArmState[i]:=SlaveArmState_Standby;
			END_IF
		
		// instrument retract
		SlaveArmState_InstruRetract:
			// to Adjust
			IF (m_slaveArms[i].adjustOn) THEN
				m_nextSlaveArmState[i]:=SlaveArmState_Adjust;
			// to standby
			ELSIF m_armCtrl[i].isFinished THEN
				m_nextSlaveArmState[i]:=SlaveArmState_Standby;
			END_IF
		
		// instrument invasion
		SlaveArmState_InstruInvasion:
			// to instrument retract
			IF NOT m_slaveArms[i].instruOn THEN
				m_nextSlaveArmState[i]:=SlaveArmState_InstruRetract;
				m_slaveArms[i].recordInstruDepth();
			// to Adjust
			elsIF (m_slaveArms[i].adjustOn) THEN
				m_nextSlaveArmState[i]:=SlaveArmState_Adjust;
			// to instrument ready
			ELSIF m_armCtrl[i].isFinished THEN
				// to endoscope ready
				IF InstruType_endoscope = m_slaveArms[i].instrument.onChipData.m_Instrutype THEN
					m_nextSlaveArmState[i]:=SlaveArmState_ScopeReady;
				// to instrument ready
				ELSE
					m_nextSlaveArmState[i]:=SlaveArmState_InstruReady;
				END_IF
			END_IF
		
		// arm disable
		SlaveArmState_Disable:
			IF NOT(i_slavesInputDataPool.m_UIData.m_slaveArmDisableFlag[i]) THEN
				// to standby
				IF m_selfCheckPass[i] THEN
					m_nextSlaveArmState[i] :=SlaveArmState_Standby;
				// to init
				ELSE
					m_nextSlaveArmState[i] :=SlaveArmState_Init;
				END_IF
			END_IF
	END_CASE
	
	// control is forbidden if setup arm is not in Hold
	IF SetupArmState_Hold <> i_slavesInputDataPool.m_setupStatus.m_armState[i] AND
		(SlaveArmState_InstruReady = m_nextSlaveArmState[i] OR SlaveArmState_MasterSlave = m_nextSlaveArmState[i]
		 OR SlaveArmState_ScopeReady = m_nextSlaveArmState[i] OR SlaveArmState_EndoScope = m_nextSlaveArmState[i]) THEN
		m_nextSlaveArmState[i]:=SlaveArmState_Standby;
	END_IF
	
	// to cart
	IF i_slavesInputDataPool.m_cartStatus.m_inMotion AND m_nextSlaveArmState[i] > SlaveArmState_Init THEN
		m_nextSlaveArmState[i] := SlaveArmState_Cart;
	END_IF
	
	// arm disable
	IF i_slavesInputDataPool.m_UIData.m_slaveArmDisableFlag[i] THEN
		m_nextSlaveArmState[i] := SlaveArmState_Disable;
	// error check
	ELSIF i_slavesInputDataPool.m_safetyData.m_slaveErrFlag[i] THEN
		m_nextSlaveArmState[i]:=SlaveArmState_Error;
	END_IF
END_FOR
END_METHOD

END_FUNCTION_BLOCK

// ---- FBs_SlaveControllers/FB_SlaveCtrlInit.TcPOU
// Brief: Slave Arm Init
FUNCTION_BLOCK PUBLIC FB_SlaveCtrlInit EXTENDS FB_SlaveArmCtrlBase
VAR_INPUT
END_VAR
VAR_OUTPUT
END_VAR
VAR
	m_initState :INT :=0;
END_VAR

// override this function in each exact controller
METHOD PROTECTED calcCmdJntPos : BOOL
VAR_IN_OUT CONSTANT
	i_endoscopePose : ST_Frame;
	i_masterStatus :ST_MasterStatus;
	i_setupStatus: ST_SetupStatus;
	i_slaveArm :FB_SlaveArm;
END_VAR

VAR 
	curInstruDepth:LREAL;
END_VAR
IF m_timePeriod > 1.0 THEN
	m_isFinished := true;
END_IF
END_METHOD

METHOD PUBLIC init : BOOL
VAR_IN_OUT CONSTANT
	i_slaveArm	:FB_SlaveArm;
END_VAR
VAR_IN_OUT 
	r_slaveArmCtrlCmd :ST_SlaveArmCtrlCmds;
END_VAR

VAR
	i:INT;
END_VAR
SUPER^.Init(i_slaveArm,r_slaveArmCtrlCmd);
m_jntEnableFlag:=g_zeroVec8i;

// update commands to arm
copyCmds(r_slaveArmCtrlCmd);
END_METHOD

END_FUNCTION_BLOCK

// ---- Mains/SetupArmControl.TcPOU
PROGRAM SetupArmControl
VAR
	// flag to init robot
	m_robotInit :BOOL :=FALSE;
	
	// wait time before robot init  for ethercat to be statble 
	m_robotInitWaitTime : LREAL:=0;
	
	// setup robot
	m_setupRobot:FB_SetupRobot;
	
	// setup robot information
	m_setupStatus AT %Q* :ST_SetupStatus;
	
	// setup robot joint data
	m_setupJointsData AT %Q* :ST_SetupJointData;
	
	// all data from other tasks and controller 
	m_setupInputDataPool : ST_SetupInputDataPool;
	
END_VAR

// wait communication to be stable
IF(m_robotInitWaitTime<g_robotInitWaitTime) THEN
	m_robotInitWaitTime := m_robotInitWaitTime+g_setupArmCtrlCycleTime;
	RETURN;
END_IF

// robot init
IF m_robotInit =FALSE THEN
	m_setupRobot.Init();
	m_robotInit:=TRUE;
END_IF

// robot run
m_setupRobot.run(m_setupInputDataPool);

// update data pool
m_setupRobot.getStatus(m_setupStatus,m_setupJointsData);

END_PROGRAM

// ---- Mains/SlaveArmControl.TcPOU
PROGRAM SlaveArmControl
VAR
	// master robot data, input from master controller box
	m_masterRobotData AT %I* : MSCommu_MasterStatus;
	
	// all data from other tasks and controller 
	m_slaveInputDataPool : ST_SlaveInputDataPool;
		
	// slave robot data, ouput to master controller box
	m_slaveRobotData AT %Q* :MSCommu_slaveStatus;
	
	// slave robot status, including arm status and cartesian data, output to other tasks
	m_slaveStatus AT%Q* :ST_slaveStatus;
	
	// slave robot joint data, output to other tasks
	m_slaveJointsData AT %Q* :ST_slaveJointData;
	
	// flag to init robot
	m_robotInit :BOOL :=FALSE;
	
	// wait time before robot init  for ethercat to be statble 
	m_robotInitWaitTime : LREAL:=0;
	
	// slave robot
	m_slaveRobot:FB_SlaveRobot;

	// code execute time measure
	m_codeTime : Profiler;
	

END_VAR

m_codeTime(START:=TRUE, RESET:=TRUE);

// wait communication to be stable
IF(m_robotInitWaitTime<g_robotInitWaitTime) THEN
	m_robotInitWaitTime := m_robotInitWaitTime+g_slaveArmCtrlCycleTime;
	RETURN;
END_IF

// robot init
IF m_robotInit =FALSE THEN
	m_slaveRobot.Init();
	m_robotInit:=TRUE;
END_IF

// input from UI
UIInputProcess();

// master input data cast
masterInputDataCast(m_masterRobotData, m_slaveInputDataPool.m_masterStatus);

// robot run
m_slaveRobot.run(m_slaveInputDataPool);

// update data pool
m_slaveRobot.getStatus(m_slaveStatus,m_slaveJointsData);

// slave output data cast
slaveOutputDataCast(m_slaveInputDataPool.m_setupStatus, m_slaveStatus, m_slaveRobotData);

// output to UI
UIOutputProcess();

m_codeTime(START:=FALSE);

// convert from MSCommu_Mastertatus for master-slave communication to local ST_MasterStatus for control
METHOD masterInputDataCast : BOOL
VAR_IN_OUT CONSTANT
	masterInputData:MSCommu_MasterStatus;
END_VAR
VAR_IN_OUT
	masterStatus :ST_MasterStatus;
END_VAR

VAR
	i : INT;
END_VAR
masterStatus.m_masterHeartBeat := masterInputData.m_heartBeat;
masterStatus.m_motionScale := masterInputData.m_motionScale;
masterStatus.m_slaveSelfCheckFlag := masterInputData.m_slaveSelfCheckFlag;

FOR i:=1 TO g_mArmNum DO
	masterStatus.m_armState[i] := masterInputData.m_armState[i];
	masterStatus.m_teleSlaveArmIdx[i] :=masterInputData.m_teleSlaveArmIdx[i];
	masterStatus.m_gripAngle[i] := masterInputData.m_gripAngle[i];
	masterStatus.m_curArmPose[i].m_pos := masterInputData.m_curArmPose[i].m_pos;
	masterStatus.m_curArmPose[i].m_rot := masterInputData.m_curArmPose[i].m_rot;
	masterStatus.m_curArmTwist[i] :=masterInputData.m_curArmTwist[i];
END_FOR
END_METHOD

// convert from local ST_SlaveStatus for control to MSCommu_SlaveStatus for master-slave communication
METHOD slaveOutputDataCast : BOOL
VAR_IN_OUT CONSTANT
	setupStatus :ST_SetupStatus;
	slaveStatus :ST_SlaveStatus;
END_VAR
VAR_IN_OUT 
	slaveOutputData : MSCommu_SlaveStatus;
END_VAR

VAR
	slavePoseInCart, slavePoseInScope:ST_Frame;
	tmpFrame :ST_Frame;
	i :INT;
END_VAR
// Slave heart beat
IF slaveOutputData.m_heartBeat > 10 THEN
	slaveOutputData.m_heartBeat :=0;
ELSE
	slaveOutputData.m_heartBeat :=slaveOutputData.m_heartBeat+1;
END_IF

slaveOutputData.m_seflCheckPass:= slaveStatus.m_selfCheckPass[1] AND slaveStatus.m_selfCheckPass[2] AND slaveStatus.m_selfCheckPass[3] AND slaveStatus.m_selfCheckPass[4];

slaveOutputData.m_endoscopeMounted :=slaveStatus.m_endoscopeMounted;
slaveOutputData.m_endoscopePose.m_pos :=slaveStatus.m_endoscopePose.m_pos;
slaveOutputData.m_endoscopePose.m_rot :=slaveStatus.m_endoscopePose.m_rot;
FOR i:= 1 TO g_sArmNum DO
	slaveOutputData.m_armState[i] := slaveStatus.m_armState[i];
	slaveOutputData.m_instruStauts[i].m_fingerAngle := slaveStatus.m_instruStauts[i].m_fingerAngle;
	slaveOutputData.m_instruStauts[i].m_ready := slaveStatus.m_instruStauts[i].m_ready;
	slaveOutputData.m_instruStauts[i].m_type := slaveStatus.m_instruStauts[i].m_type;

	slavePoseInCart := transform(setupStatus.m_curEndPose[i], slaveStatus.m_curArmPose[i]);
	tmpFrame :=invFrame(slaveStatus.m_endoscopePose);
	slavePoseInScope := transform(tmpFrame, slavePoseInCart);
	slaveOutputData.m_curArmPose[i].m_pos :=slavePoseInScope.m_pos;
	slaveOutputData.m_curArmPose[i].m_rot :=slavePoseInScope.m_rot;
	slaveOutputData.m_masterSlavePoseError[i] :=slaveStatus.m_masterSlavePoseError[i];
END_FOR
END_METHOD

// tranform data from UI(global variable write by ADS) to ST_UIData
METHOD UIInputProcess : BOOL
VAR_INPUT
END_VAR
VAR
	i:int;
END_VAR
// arm disable
FOR i:=1 TO g_sArmNum DO 
	m_slaveInputDataPool.m_UIData.m_slaveArmDisableFlag[i]:= FALSE;
END_FOR
IF GVL_com_upper_PC.slaver_arm_disable >0 AND GVL_com_upper_PC.slaver_arm_disable<= g_sArmNum THEN
	m_slaveInputDataPool.m_UIData.m_slaveArmDisableFlag[GVL_com_upper_PC.slaver_arm_disable]:= TRUE;
END_IF
END_METHOD

METHOD UIOutputProcess : BOOL
VAR_INPUT
END_VAR
VAR
	i : INT;
END_VAR
//TODO
//control software version
GVL_com_upper_PC.version:='1(1.0.0.1)';

GVL_com_upper_PC.state_machine.Arm1_state_machine := m_slaveRobot.m_slaveArmState[1];
GVL_com_upper_PC.state_machine.Arm2_state_machine := m_slaveRobot.m_slaveArmState[2];
GVL_com_upper_PC.state_machine.Arm3_state_machine := m_slaveRobot.m_slaveArmState[3];
GVL_com_upper_PC.state_machine.Arm4_state_machine := m_slaveRobot.m_slaveArmState[4];
END_METHOD

END_PROGRAM

// ---- Mains/RobotDynamics.TcPOU
PROGRAM RobotDynamics

VAR
	// slave robot arms joint data
	m_slaveJointsData AT %I* :ST_SlaveJointData;
	
	// setup joint5 position
	m_setupJointData AT %I* :ST_SetupJointData;
	
	// instrument info
	m_instruInfo AT %I* :ARRAY[1..g_sArmNum] OF ST_InstruStatus;
	
	// dynamic output
	m_slaveDynaData AT %Q* : ST_SlaveDynaData;
	m_setupJnt3Gravity AT %Q* : ARRAY[1..g_sArmNum] OF LREAL;
	m_setupJnt5Gravity AT %Q* : ARRAY[1..g_sArmNum] OF LREAL;
	
	// flag to init robot dynamic model
	m_robotDynaInit :BOOL :=FALSE;
	
	// grivity model block
	m_slaveGravityModel :ARRAY[1..g_sArmNum] OF FB_SlaveGravity;
	m_setupGravityModel :ARRAY[1..g_sArmNum] OF FB_SetupGravity;
	

	// code execute time measure
	m_codeTime : Profiler;
	
	// tmp variables
	i: INT;
	
END_VAR

m_codeTime(START:=TRUE, RESET:=TRUE);

// robot dynamic model init
IF m_robotDynaInit =FALSE THEN
	FOR i:=1 TO g_sArmNum DO
		m_slaveGravityModel[i].Init(i);
		m_setupGravityModel[i].init(i);
	END_FOR

	m_robotDynaInit:=TRUE;
END_IF

// run gravity model
FOR i:=1 TO g_sArmNum DO
//	m_setupJointData.m_curJntPos[i][5]:=pi/2;
	m_slaveDynaData.m_gravity[i]:=m_slaveGravityModel[i].run(m_setupJointData.m_curJntPos[i][5], m_slaveJointsData.m_curJntPos[i],m_instruInfo[i]);
	m_setupGravityModel[i].run(m_setupJointData.m_curJntPos[i], m_slaveJointsData.m_curJntPos[i],m_instruInfo[i], o_jnt3Gravity=> m_setupJnt3Gravity[i], o_jnt5Gravity=> m_setupJnt5Gravity[i]);
END_FOR


m_codeTime(START:=FALSE);

END_PROGRAM

// ---- SafetyCheck/FB_SlaveArmCheck.TcPOU
FUNCTION_BLOCK FB_SlaveArmCheck
VAR_INPUT
END_VAR
VAR_OUTPUT
END_VAR
VAR
	// final arm error flag
	m_armErrFlag :ARRAY[1..g_sArmNum] OF BOOL:=[4(FALSE)];
	
	// cartesian pose error flag
	m_cartPoseErrFlag :ARRAY[1..g_sArmNum] OF BOOL;
	m_cartPoseErrCounts:ARRAY[1..g_sArmNum] OF INT;
	m_cartPosErr :ARRAY[1..g_sArmNum] OF Vec3d;	// cartesian position error
	m_cartOriErr:ARRAY[1..g_sArmNum] OF  Vec3d;	// cartesian rotation angle (angle  * axis)
	
	// joint control error flag
	m_jntCtrlErrFlag :ARRAY[1..g_sArmNum] OF Vec8b;
	m_jntCtrlErrCounts :ARRAY[1..g_sArmNum] OF Vec8i;
	m_jntCtrlErr:ARRAY[1..g_sArmNum]  OF Vec8d;		// joint position control error
	
	// joint encoder error flag
	m_jntEncErrFlag :ARRAY[1..g_sArmNum] OF Vec8b;
	m_jntEncErrCounts :ARRAY[1..g_sArmNum] OF Vec8i ;
	m_jntEncErr:ARRAY[1..g_sArmNum]  OF Vec8d;		// motor and joint encoder error
	
	// joint velocity error flag
	m_jntVelErrFlag :ARRAY[1..g_sArmNum] OF Vec8b;
	m_jntVelErrCounts :ARRAY[1..g_sArmNum] OF Vec8i;
	
	// joint position limit error flag
	m_jntLimitErrFlag :ARRAY[1..g_sArmNum] OF Vec8b;
	m_jntLimitErrCounts :ARRAY[1..g_sArmNum] OF Vec8i;

END_VAR

METHOD check : BOOL
VAR_IN_OUT CONSTANT
	i_slaveStatus : ST_SlaveStatus;
	i_slaveJointData :ST_SlaveJointData;
END_VAR
VAR_OUTPUT
	o_errorFlag :ARRAY[1..g_sArmNum] OF BOOL ;
END_VAR

VAR
	i ,j:INT ;
END_VAR
// calculate error
FOR i:=1 TO g_sArmNum DO 
	// stop check if arm is already in error state
	IF m_armErrFlag[i] OR i_slaveStatus.m_armState[i]=SlaveArmState_Error THEN 
		CONTINUE;
	END_IF
	
	// only check cartesion pose error in master-slave mode
	m_cartPoseErrFlag[i]:=FALSE;
	IF  SlaveArmState_MasterSlave = i_slaveStatus.m_armState[i] THEN 
		m_cartPoseErrFlag[i]:=poseErrCheck(i_slaveStatus.m_cmdArmPose[i],  i_slaveStatus.m_curArmPose[i],
											m_cartPoseErrCounts[i], m_cartPosErr[i], m_cartOriErr[i]);
	END_IF
	
	// joint control error
	m_jntCtrlErrFlag[i]:=jntCtrlErrCheck(i_slaveJointData.m_cmdJntPos[i], i_slaveJointData.m_curJntPos[i],
										m_jntCtrlErrCounts[i], m_jntCtrlErr[i]);
	
	// encoder error
	m_jntEncErrFlag[i]:=jntEncErrCheck(i_slaveJointData.m_curMotorPos[i], i_slaveJointData.m_curLinkPos[i],
										m_jntEncErrCounts[i], m_jntEncErr[i]);
										
	// joint limit error
	m_jntLimitErrFlag[i]:=jntLimitErrCheck(i_slaveJointData.m_curJntPos[i],m_jntLimitErrCounts[i]);
										
	// final arm error status check
	IF  m_cartPoseErrFlag[i] THEN
		m_armErrFlag[i]:=TRUE;
		CONTINUE;
	END_IF
	
	FOR j:=1 TO g_sJntNum DO 
		IF m_jntCtrlErrFlag[i][j] OR m_jntEncErrFlag[i][j] OR m_jntVelErrFlag[i][j] OR m_jntLimitErrFlag[i][j] THEN
			m_armErrFlag[i]:=TRUE;
			EXIT;
		END_IF
	END_FOR
	
END_FOR

o_errorFlag:=m_armErrFlag;
END_METHOD

METHOD jntCtrlErrCheck : Vec8b
VAR_INput
	i_cmdJntPos : Vec8d;
	i_curJntPos : Vec8d;
END_VAR
VAR_IN_OUT
	r_errCount:Vec8i;
	r_jntCtrlErr :Vec8d;
END_VAR

VAR
	i :INT;
	err:Vec8d;
END_VAR
vecSub(i_cmdJntPos,i_curJntPos,  err);
r_jntCtrlErr:=err;

// joint error check
//NOTE: only check the first three joints.
FOR i:=1 TO 3 DO 
	IF  ABS(r_jntCtrlErr[i]) > g_slaveMaxJntCtrlErr[i] THEN
		r_errCount[i]:=r_errCount[i]+1;
	ELSE
		r_errCount[i] :=0;	
	END_IF
	jntCtrlErrCheck[i]:= r_errCount[i]>=g_faultTriggerCounts;
END_FOR
END_METHOD

METHOD jntEncErrCheck : Vec8b
VAR_INput
	i_motorJntPos : Vec8d;
	i_linkJntPos : Vec8d;
END_VAR
VAR_IN_OUT
	r_errCount:Vec8i;
	r_jntEncErr :Vec8d;
END_VAR

VAR
	i :INT;
	err:Vec8d;
END_VAR
vecSub(i_motorJntPos,i_linkJntPos,  err);
r_jntEncErr:=err;

// joint error check
FOR i:=1 TO g_sJntNum DO 
	IF  ABS(r_jntEncErr[i]) > g_slaveMaxJntCtrlErr[i] THEN
		r_errCount[i]:=r_errCount[i]+1;
	ELSE
		r_errCount[i] :=0;
	END_IF
	jntEncErrCheck[i]:= r_errCount[i]>=g_faultTriggerCounts;
END_FOR

// NOTE: power box joints are easy to trigger encoder error during instrument mount, so this part is diabled now
FOR i:=4 TO g_sJntNum DO
	jntEncErrCheck[i] := false;
END_FOR
END_METHOD

METHOD jntLimitErrCheck : Vec8b
VAR_INput
	i_curJntPos : Vec8d;
END_VAR
VAR_IN_OUT
	r_errCount:Vec8i;
END_VAR

VAR
	i :INT;
END_VAR
// joint limit check
//NOTE: only check the first three joints.
FOR i:=1 TO 3 DO 
	IF  i_curJntPos[i] > GVL_SlaveMotorParameters.g_maxJntPos[i] + g_slaveJntPosLimitBuffer[i] OR
		i_curJntPos[i] < GVL_SlaveMotorParameters.g_minJntPos[i] - g_slaveJntPosLimitBuffer[i] THEN
		r_errCount[i]:=r_errCount[i]+1;
	ELSE
		r_errCount[i] :=0;	
	END_IF
	jntLimitErrCheck[i]:= r_errCount[i]>=g_faultTriggerCounts;
END_FOR
END_METHOD

METHOD poseErrCheck : BOOL
VAR_INPUT
	i_cmdPose : ST_Frame;
	i_curPose :ST_Frame;
END_VAR
VAR_IN_OUT
	r_errCount:INT;
	r_posErr :Vec3d;
	r_oriErr :Vec3d;
END_VAR

VAR
	posErr,oriErr:Vec3d;
	matT,rotErr:Mat3d;
	errAngle :LREAL;
	errAxis :Vec3d;
END_VAR
vecSub(i_cmdPose.m_pos, i_curPose.m_pos,posErr);
r_posErr:=posErr;

matTranspose(i_cmdPose.m_rot, matT);
matMultiply(matT,i_curPose.m_rot, rotErr);
rot2AngAxis(rotErr, angle=>errAngle, axis=>errAxis);
vecMultiNum(errAxis, errAngle,oriErr);
r_oriErr:=oriErr;
	
IF  norm(posErr)>g_maxCartPosErr OR norm(oriErr)> g_maxCartOriErr THEN
	r_errCount:= r_errCount +1;
ELSE 
	r_errCount:=0;
END_IF
poseErrCheck:= r_errCount >= g_faultTriggerCounts;
END_METHOD

END_FUNCTION_BLOCK
